METHOD PUBLIC PreExecutionCheck
VAR_INPUT
	Check : I_PreExecutionChecks;
END_VAR
Check.IsTrue(ipSrcImage.IsValid, 'ipSrcImage must contain an image');
Check.IsTrue(ipSrcImage.HasChannelCount(1), 'ipSrcImage must have 1 channel');
Check.IsTrue(ipSrcImage.IsPixelDepth(8), 'ipSrcImage must have 8 bit pixel depth');
Check.IsTrue((fMaxValue.Value >= 0.0), 'fMaxValue must be greater than or equal to 0');
Check.IsTrue((fMaxValue.Value <= 255.0), 'fMaxValue must be less than or equal to 255');
Check.IsTrue((eThresholdType.Value = ETcVnThresholdType.TCVN_TT_BINARY OR 
              eThresholdType.Value = ETcVnThresholdType.TCVN_TT_BINARY_INV), 'eThresholdType must be TCVN_TT_BINARY or TCVN_TT_BINARY_INV');
Check.IsTrue(nBlockSize.Value >= 3, 'nBlockSize must be greater than or equal to 3');
Check.IsTrue(nBlockSize.IsOdd, 'nBlockSize must be an odd number');
END_METHOD

END_FUNCTION_BLOCK

// ---- Nodes/Image Segmentation/Node_F_VN_SauvolaThreshold.TcPOU
{attribute 'linkalways'} 
{attribute 'no_explicit_call' := 'This FB is a CLASS and must be accessed using methods or properties'}
{attribute 'enable_dynamic_creation'}
FUNCTION_BLOCK Node_F_VN_SauvolaThreshold EXTENDS VisionNode
VAR
	ipSrcImage : _ITcVnImage;
    pipDestImage : _ITcVnImage;
    nBlockSize : _UDINT(3);
    fParamK : _LREAL(0.0);
    fMaxSigma : _LREAL(0.0);
    eThresholdType : _ETcVnThresholdType(ETcVnThresholdType.TCVN_TT_BINARY);
    hrPrev : _HRESULT(S_OK);
	hresult : _HRESULT(S_OK);
END_VAR

METHOD PUBLIC  Clone : I_Node
VAR
	pNode : POINTER TO Node_F_VN_SauvolaThreshold;
END_VAR
pNode := __NEW(Node_F_VN_SauvolaThreshold);
Clone := pNode^;
END_METHOD

METHOD FB_init : BOOL
VAR_INPUT
	bInitRetains : BOOL; // if TRUE, the retain variables are initialized (warm start / cold start)
	bInCopyCode : BOOL;  // if TRUE, the instance afterwards gets moved into the copy code (online change)
END_VAR
AddInput('ipSrcImage', ipSrcImage);
AddParameter('nBlockSize', nBlockSize);
AddParameter('fParamK', fParamK);
AddParameter('fMaxSigma', fMaxSigma);
AddParameter('eThresholdType', eThresholdType);
AddInput('hrPrev', hrPrev);
AddOutput('pipDestImage', pipDestImage);
AddOutput('hresult', hresult);
END_METHOD

METHOD PROTECTED OnExecute
hresult.Value := F_VN_SauvolaThreshold(
	ipSrcImage := ipSrcImage.Value,
	pipDestImage := pipDestImage.Value,
    nBlockSize := nBlockSize.Value,
    fParamK := fParamK.Value,
    fMaxSigma := fMaxSigma.Value,
    eThresholdType := eThresholdType.Value,
	hrPrev := hrPrev.Value);
END_METHOD

METHOD PUBLIC PreExecutionCheck
VAR_INPUT
	Check : I_PreExecutionChecks;
END_VAR
Check.IsTrue(ipSrcImage.IsValid, 'ipSrcImage must contain an image');
Check.IsTrue(ipSrcImage.HasChannelCount(1), 'ipSrcImage must have 1 channel');

Check.IsTrue((ipSrcImage.IsPixelDepth(8) OR
              ipSrcImage.IsPixelDepth(16) OR
              ipSrcImage.IsPixelDepth(32) OR
              ipSrcImage.IsPixelDepth(6432)), 'ipSrcImage must have 8, 16, 32, or 64 bit pixel depth');

Check.IsTrue(nBlockSize.IsOdd, 'nBlockSize must be an odd number');
Check.IsTrue(nBlockSize.Value >= 3, 'nBlockSize must be greater than or equal to 3');

Check.IsTrue((fParamK.Value >= 0.0), 'fMaxValue must be greater than or equal to 0');
Check.IsTrue((fParamK.Value <= 1.0), 'fMaxValue must be less than or equal to 1');

Check.IsTrue((fMaxSigma.Value >= 0.0), 'fMaxValue must be greater than or equal to 0');

Check.IsTrue((eThresholdType.Value = ETcVnThresholdType.TCVN_TT_BINARY OR 
              eThresholdType.Value = ETcVnThresholdType.TCVN_TT_BINARY_INV), 'eThresholdType must be TCVN_TT_BINARY or TCVN_TT_BINARY_INV');
END_METHOD

END_FUNCTION_BLOCK

// ---- Nodes/Image Segmentation/Node_F_VN_DoubleThreshold.TcPOU
{attribute 'linkalways'} 
{attribute 'no_explicit_call' := 'This FB is a CLASS and must be accessed using methods or properties'}
{attribute 'enable_dynamic_creation'}
FUNCTION_BLOCK Node_F_VN_DoubleThreshold EXTENDS VisionNode
VAR
	ipSrcImage : _ITcVnImage;
    ipDestImage : _ITcVnImage;
    fLowThreshold : _LREAL(0.0);
    fHighThreshold : _LREAL(0.0);
    fMaxValue : _LREAL(0.0);
    hrPrev : _HRESULT(S_OK);
	hresult : _HRESULT(S_OK);
END_VAR

METHOD PUBLIC  Clone : I_Node
VAR
	pNode : POINTER TO Node_F_VN_DoubleThreshold;
END_VAR
pNode := __NEW(Node_F_VN_DoubleThreshold);
Clone := pNode^;
END_METHOD

METHOD FB_init : BOOL
VAR_INPUT
	bInitRetains : BOOL; // if TRUE, the retain variables are initialized (warm start / cold start)
	bInCopyCode : BOOL;  // if TRUE, the instance afterwards gets moved into the copy code (online change)
END_VAR
AddInput('ipSrcImage', ipSrcImage);
AddParameter('fLowThreshold', fLowThreshold);
AddParameter('fHighThreshold', fHighThreshold);
AddParameter('fMaxValue', fMaxValue);
AddInput('hrPrev', hrPrev);
AddOutput('ipDestImage', ipDestImage);
AddOutput('hresult', hresult);
END_METHOD

METHOD PROTECTED OnExecute
hresult.Value := F_VN_DoubleThreshold(
	ipSrcImage := ipSrcImage.Value,
	ipDestImage := ipDestImage.Value,
    fLowThreshold := fLowThreshold.Value,
    fHighThreshold := fHighThreshold.Value,
    fMaxValue := fMaxValue.Value,
	hrPrev := hrPrev.Value);
END_METHOD

METHOD PUBLIC PreExecutionCheck
VAR_INPUT
	Check : I_PreExecutionChecks;
END_VAR
VAR
    pixelFormat : TcVnPixelFormat;
END_VAR
Check.IsTrue(ipSrcImage.IsValid, 'ipSrcImage must contain an image');
Check.IsTrue(ipSrcImage.HasChannelCount(1), 'ipSrcImage must have 1 channel');
Check.IsTrue((ipSrcImage.IsPixelDepth(8) OR
              ipSrcImage.IsPixelDepth(16) OR
              ipSrcImage.IsPixelDepth(32) OR
              ipSrcImage.IsPixelDepth(64)), 'ipSrcImage must have 8, 16, 32, or 64 bit pixel depth');

ipSrcImage.TryGetPixelFormat(pixelFormat);
Check.IsTrue(IsMaxValueCompatibleWithPixelDepth(fMaxValue.Value, pixelFormat.nElementSize), 'fMaxValue is not compatible with pixel depth');
END_METHOD

END_FUNCTION_BLOCK

// ---- Nodes/Image Segmentation/Node_F_VN_WatershedSegmentationExp.TcPOU
{attribute 'linkalways'} 
{attribute 'no_explicit_call' := 'This FB is a CLASS and must be accessed using methods or properties'}
{attribute 'enable_dynamic_creation'}
FUNCTION_BLOCK Node_F_VN_WatershedSegmentationExp EXTENDS VisionNode
VAR
	ipSrcImage : _ITcVnImage;
    ipDestImage : _ITcVnImage;
    ipMarkers : _ITcVnImage;
    hrPrev : _HRESULT(S_OK);
	hresult : _HRESULT(S_OK);
END_VAR

METHOD PUBLIC  Clone : I_Node
VAR
	pNode : POINTER TO Node_F_VN_WatershedSegmentationExp;
END_VAR
pNode := __NEW(Node_F_VN_WatershedSegmentationExp);
Clone := pNode^;
END_METHOD

METHOD FB_init : BOOL
VAR_INPUT
	bInitRetains : BOOL; // if TRUE, the retain variables are initialized (warm start / cold start)
	bInCopyCode : BOOL;  // if TRUE, the instance afterwards gets moved into the copy code (online change)
END_VAR
AddInput('ipSrcImage', ipSrcImage);
AddInput('ipMarkers', ipMarkers);
AddInput('hrPrev', hrPrev);
AddOutput('ipDestImage', ipDestImage);
AddOutput('hresult',hresult);
END_METHOD

METHOD PROTECTED OnExecute
hresult.Value := F_VN_WatershedSegmentationExp(
	ipSrcImage := ipSrcImage.Value,
	ipDestImage := ipDestImage.Value,
    ipMarkers := ipMarkers.Value,
	hrPrev := hrPrev.Value);
END_METHOD

METHOD PUBLIC PreExecutionCheck
VAR_INPUT
	Check : I_PreExecutionChecks;
END_VAR
Check.IsTrue(ipSrcImage.IsValid, 'ipSrcImage must contain an image');
Check.IsTrue(ipSrcImage.HasChannelCount(3), 'ipSrcImage must have 3 channels');
Check.IsTrue(ipSrcImage.IsPixelDepth(8), 'ipSrcImage must have 8 bit pixel depth');
Check.IsTrue(ipMarkers.IsValid, 'ipMarkers must contain an image');
Check.IsTrue(ipMarkers.HasChannelCount(1), 'ipMarkers must have 1 channel');
Check.IsTrue(ipMarkers.IsPixelDepth(32), 'ipMarkers must have DINT 32 bit pixel depth');
END_METHOD

END_FUNCTION_BLOCK

// ---- Nodes/Image Segmentation/Node_F_VN_CheckColorRange.TcPOU
{attribute 'linkalways'} 
{attribute 'no_explicit_call' := 'This FB is a CLASS and must be accessed using methods or properties'}
{attribute 'enable_dynamic_creation'}
FUNCTION_BLOCK Node_F_VN_CheckColorRange EXTENDS VisionNode
VAR
	ipSrcImage : _ITcVnImage;
    ipDestImage : _ITcVnImage;
    aLowerBounds : _TcVnVector4_LREAL;
    aUpperBounds : _TcVnVector4_LREAL;
    hrPrev : _HRESULT(S_OK);
	hresult : _HRESULT(S_OK);
END_VAR

METHOD PUBLIC  Clone : I_Node
VAR
	pNode : POINTER TO Node_F_VN_CheckColorRange;
END_VAR
pNode := __NEW(Node_F_VN_CheckColorRange);
Clone := pNode^;
END_METHOD

METHOD FB_init : BOOL
VAR_INPUT
	bInitRetains : BOOL; // if TRUE, the retain variables are initialized (warm start / cold start)
	bInCopyCode : BOOL;  // if TRUE, the instance afterwards gets moved into the copy code (online change)
END_VAR
AddInput('ipSrcImage', ipSrcImage);
AddInput('aLowerBounds', aLowerBounds);
AddInput('aUpperBounds', aUpperBounds);
AddInput('hrPrev', hrPrev);
AddOutput('ipDestImage', ipDestImage);
AddOutput('hresult', hresult);
END_METHOD

METHOD PROTECTED OnExecute
hresult.Value := F_VN_CheckColorRange(
	ipSrcImage := ipSrcImage.Value,
	ipDestImage := ipDestImage.Value,
    aLowerBounds := aLowerBounds.Value,
    aUpperBounds := aUpperBounds.Value,
	hrPrev := hrPrev.Value);
END_METHOD

METHOD PUBLIC PreExecutionCheck
VAR_INPUT
	Check : I_PreExecutionChecks;
END_VAR
Check.IsTrue(ipSrcImage.IsValid, 'ipSrcImage must contain an image');
END_METHOD

END_FUNCTION_BLOCK

// ---- Nodes/Image Segmentation/Node_F_VN_AdaptiveThreshold.TcPOU
{attribute 'linkalways'} 
{attribute 'no_explicit_call' := 'This FB is a CLASS and must be accessed using methods or properties'}
{attribute 'enable_dynamic_creation'}
FUNCTION_BLOCK Node_F_VN_AdaptiveThreshold EXTENDS VisionNode
VAR
	ipSrcImage : _ITcVnImage;
    ipDestImage : _ITcVnImage;
    fMaxValue : _LREAL(0.0);
    hrPrev : _HRESULT(S_OK);
	hresult : _HRESULT(S_OK);
END_VAR

METHOD PUBLIC  Clone : I_Node
VAR
	pNode : POINTER TO Node_F_VN_AdaptiveThreshold;
END_VAR
pNode := __NEW(Node_F_VN_AdaptiveThreshold);
Clone := pNode^;
END_METHOD

METHOD FB_init : BOOL
VAR_INPUT
	bInitRetains : BOOL; // if TRUE, the retain variables are initialized (warm start / cold start)
	bInCopyCode : BOOL;  // if TRUE, the instance afterwards gets moved into the copy code (online change)
END_VAR
AddInput('ipSrcImage', ipSrcImage);
AddParameter('fMaxValue', fMaxValue);
AddInput('hrPrev', hrPrev);
AddOutput('ipDestImage', ipDestImage);
AddOutput('hresult', hresult);
END_METHOD

METHOD PROTECTED OnExecute
hresult.Value := F_VN_AdaptiveThreshold(
	ipSrcImage := ipSrcImage.Value,
	ipDestImage := ipDestImage.Value,
    fMaxValue := fMaxValue.Value,
	hrPrev := hrPrev.Value);
END_METHOD

METHOD PUBLIC PreExecutionCheck
VAR_INPUT
	Check : I_PreExecutionChecks;
END_VAR
Check.IsTrue(ipSrcImage.IsValid, 'ipSrcImage must contain an image');
Check.IsTrue(ipSrcImage.HasChannelCount(1), 'ipSrcImage must have 1 channel');
Check.IsTrue(ipSrcImage.IsPixelDepth(8), 'ipSrcImage must have 8 bit pixel depth');
Check.IsTrue((fMaxValue.Value >= 0.0), 'fMaxValue must be greater than or equal to 0');
Check.IsTrue((fMaxValue.Value <= 255.0), 'fMaxValue must be less than or equal to 255');
END_METHOD

END_FUNCTION_BLOCK

// ---- Nodes/Image Segmentation/Node_F_VN_Threshold.TcPOU
{attribute 'linkalways'} 
{attribute 'no_explicit_call' := 'This FB is a CLASS and must be accessed using methods or properties'}
{attribute 'enable_dynamic_creation'}
FUNCTION_BLOCK Node_F_VN_Threshold EXTENDS VisionNode
VAR
	ipSrcImage : _ITcVnImage;
    ipDestImage : _ITcVnImage;
    fThreshold : _LREAL(0.0);
    fMaxValue : _LREAL(0.0);
	eThresholdType : _ETcVnThresholdType(ETcVnThresholdType.TCVN_TT_BINARY);
    hrPrev : _HRESULT(S_OK);
	hresult : _HRESULT(S_OK);
END_VAR

METHOD PUBLIC  Clone : I_Node
VAR
	pNode : POINTER TO Node_F_VN_Threshold;
END_VAR
pNode := __NEW(Node_F_VN_Threshold);
Clone := pNode^;
END_METHOD

METHOD FB_init : BOOL
VAR_INPUT
	bInitRetains : BOOL; // if TRUE, the retain variables are initialized (warm start / cold start)
	bInCopyCode : BOOL;  // if TRUE, the instance afterwards gets moved into the copy code (online change)
END_VAR
AddInput('ipSrcImage', ipSrcImage);
AddParameter('fThreshold', fThreshold);
AddParameter('fMaxValue', fMaxValue);
AddParameter('eThresholdType', eThresholdType);
AddInput('hrPrev', hrPrev);
AddOutput('ipDestImage', ipDestImage);
AddOutput('hresult',hresult);
END_METHOD

METHOD PROTECTED OnExecute
hresult.Value := F_VN_Threshold(
	ipSrcImage := ipSrcImage.Value, 
	ipDestImage := ipDestImage.Value, 
	fThreshold := fThreshold.Value, 
	fMaxValue := fMaxValue.Value, 
	eThresholdType := eThresholdType.Value, 
	hrPrev := hrPrev.Value);
END_METHOD

METHOD PUBLIC PreExecutionCheck
VAR_INPUT
	Check : I_PreExecutionChecks;
END_VAR
VAR
    dynamicThresholding : BOOL;
    pixelFormat : TcVnPixelFormat;
END_VAR
Check.IsTrue(ipSrcImage.IsValid, 'ipSrcImage must contain an image');

CASE eThresholdType.Value OF
    TCVN_TT_OTSU_BINARY,
    TCVN_TT_OTSU_BINARY_INV,
    TCVN_TT_OTSU_TRUNC,
    TCVN_TT_OTSU_TOZERO,
    TCVN_TT_OTSU_TOZERO_INV,
    TCVN_TT_TRIANGLE_BINARY,
    TCVN_TT_TRIANGLE_BINARY_INV,
    TCVN_TT_TRIANGLE_TRUNC,
    TCVN_TT_TRIANGLE_TOZERO,
    TCVN_TT_TRIANGLE_TOZERO_INV :
        dynamicThresholding := TRUE;
END_CASE

IF dynamicThresholding THEN
    Check.IsTrue(ipSrcImage.HasChannelCount(1), 'ipSrcImage must have 1 channel when using dynamic thresholding');
    Check.IsTrue(ipSrcImage.IsPixelDepth(8), 'ipSrcImage must have 8 bit pixel depth when using dynamic thresholding');
ELSE
    Check.IsTrue((ipSrcImage.HasChannelCount(1) OR ipSrcImage.HasChannelCount(3)), 'ipSrcImage must have 1 or 3 channels');
END_IF

ipSrcImage.TryGetPixelFormat(pixelFormat);
Check.IsTrue(IsMaxValueCompatibleWithPixelDepth(fMaxValue.Value, pixelFormat.nElementSize), 'fMaxValue is not compatible with pixel depth');
END_METHOD

END_FUNCTION_BLOCK

// ---- Nodes/Keypoint Features/Node_F_VN_FilterGoodMatches.TcPOU
{attribute 'linkalways'} 
{attribute 'no_explicit_call' := 'This FB is a CLASS and must be accessed using methods or properties'}
{attribute 'enable_dynamic_creation'}
FUNCTION_BLOCK Node_F_VN_FilterGoodMatches EXTENDS VisionNode
VAR
    ipMatches : _ITcVnContainer;
    ipGoodMatches : _ITcVnContainer;
    fMaxDist : _REAL(0.0);
    fMaxKnnRatio : _REAL(0.0);
    hrPrev : _HRESULT(S_OK);
	hresult : _HRESULT(S_OK);
END_VAR

METHOD PUBLIC  Clone : I_Node
VAR
	pNode : POINTER TO Node_F_VN_FilterGoodMatches;
END_VAR
pNode := __NEW(Node_F_VN_FilterGoodMatches);
Clone := pNode^;
END_METHOD

METHOD FB_init : BOOL
VAR_INPUT
	bInitRetains : BOOL; // if TRUE, the retain variables are initialized (warm start / cold start)
	bInCopyCode : BOOL;  // if TRUE, the instance afterwards gets moved into the copy code (online change)
END_VAR
AddInput('ipMatches', ipMatches);
AddParameter('fMaxDist', fMaxDist);
AddParameter('fMaxKnnRatio', fMaxKnnRatio);
AddInput('hrPrev', hrPrev);
AddOutput('ipGoodMatches', ipGoodMatches);
AddOutput('hresult',hresult);
END_METHOD

METHOD PROTECTED OnExecute
hresult.Value := F_VN_FilterGoodMatches(
    ipMatches := ipMatches.Value,
    ipGoodMatches := ipGoodMatches.Value,
    fMaxDist := fMaxDist.Value,
    fMaxKnnRatio := fMaxKnnRatio.Value,
	hrPrev:= hrPrev.Value);
END_METHOD

METHOD PUBLIC PreExecutionCheck
VAR_INPUT
	Check : I_PreExecutionChecks;
END_VAR
Check.IsTrue(ipMatches.IsValid, 'ipMatches must be a valid container');
Check.IsTrue((ipMatches.IsType(TC_GLOBAL_CONST_LIST.ContainerType_Vector_TcVnDMatch) OR
              ipMatches.IsType(TC_GLOBAL_CONST_LIST.ContainerType_Vector_Vector_TcVnDMatch)),
              'ipMatches contains incorrect type');
              
IF NOT (fMaxDist.Value = -1) THEN
    Check.IsTrue(fMaxDist.Value >= 0, 'fMaxDist must be greater than or equal to 0');
END_IF

IF NOT (fMaxKnnRatio.Value = -1) THEN
    Check.IsTrue((fMaxKnnRatio.Value >= 0 OR fMaxDist.Value <= 1), 'fMaxDist must be within 0 to 1');
END_IF
END_METHOD

END_FUNCTION_BLOCK

// ---- Nodes/Keypoint Features/Node_F_VN_FindReferenceKeyPointsInImage.TcPOU
{attribute 'linkalways'}
{attribute 'no_explicit_call' := 'This FB is a CLASS and must be accessed using methods or properties'}
{attribute 'enable_dynamic_creation'}
FUNCTION_BLOCK Node_F_VN_FindReferenceKeyPointsInImage EXTENDS VisionNode
VAR
    ipSrcKeyPoints : _ITcVnContainer;
    ipSrcDescriptors : _ITcVnImage;
    ipRefKeyPoints : _ITcVnContainer;
    ipRefDescriptors : _ITcVnImage;
    nRefImageWidth : _UDINT(0);
    nRefImageHeight : _UDINT(0);
    ipEdgePoints : _ITcVnContainer;
    fMaxDist : _REAL(-1.0);
    fMaxKnnRatio : _REAL(-1.0);
    eNormType : _ETcVnNormalizationType(ETcVnNormalizationType.TCVN_NT_HAMMING);
    hrPrev : _HRESULT(S_OK);
    aPerspectiveTransform : _TcVnMatrix3x3_LREAL;
    nNumberOfGoodMatches : _UDINT(0);
    nNumberOfInliers : _UDINT(0);
    hresult : _HRESULT(S_OK);
END_VAR

METHOD PUBLIC Clone : I_Node
VAR
    pNode : POINTER TO Node_F_VN_FindReferenceKeyPointsInImage;
END_VAR
pNode := __NEW(Node_F_VN_FindReferenceKeyPointsInImage);
Clone := pNode^;
END_METHOD

METHOD FB_init : BOOL
VAR_INPUT
    bInitRetains : BOOL;
    bInCopyCode : BOOL;
END_VAR
AddInput('ipSrcKeyPoints', ipSrcKeyPoints);
AddInput('ipSrcDescriptors', ipSrcDescriptors);
AddInput('ipRefKeyPoints', ipRefKeyPoints);
AddInput('ipRefDescriptors', ipRefDescriptors);
AddInput('nRefImageWidth', nRefImageWidth);
AddInput('nRefImageHeight', nRefImageHeight);
AddOutput('ipEdgePoints', ipEdgePoints);
AddParameter('fMaxDist', fMaxDist);
AddParameter('fMaxKnnRatio', fMaxKnnRatio);
AddParameter('eNormType', eNormType);
AddInput('hrPrev', hrPrev);
AddOutput('aPerspectiveTransform', aPerspectiveTransform);
AddOutput('nNumberOfGoodMatches', nNumberOfGoodMatches);
AddOutput('nNumberOfInliers', nNumberOfInliers);
AddOutput('hresult', hresult);
END_METHOD

METHOD PROTECTED OnExecute
VAR
    perspectiveTransform : TcVnMatrix3x3_LREAL;
    numberOfGoodMatches : UDINT;
    numberOfInliers : UDINT;
END_VAR
hresult.Value := F_VN_FindReferenceKeyPointsInImage(
    ipSrcKeyPoints := ipSrcKeyPoints.Value,
    ipSrcDescriptors := ipSrcDescriptors.Value,
    ipRefKeyPoints := ipRefKeyPoints.Value,
    ipRefDescriptors := ipRefDescriptors.Value,
    nRefImageWidth := nRefImageWidth.Value,
    nRefImageHeight := nRefImageHeight.Value,
    ipEdgePoints := ipEdgePoints.Value,
    fMaxDist := fMaxDist.Value,
    fMaxKnnRatio := fMaxKnnRatio.Value,
    eNormType := eNormType.Value,
    hrPrev := hrPrev.Value,
    aPerspectiveTransform => perspectiveTransform,
    nNumberOfGoodMatches => numberOfGoodMatches,
    nNumberOfInliers => numberOfInliers);

aPerspectiveTransform.Value := perspectiveTransform;
nNumberOfGoodMatches.Value := numberOfGoodMatches;
nNumberOfInliers.Value := numberOfInliers;
END_METHOD

METHOD PUBLIC PreExecutionCheck
VAR_INPUT
    Check : I_PreExecutionChecks;
END_VAR
Check.IsTrue(ipSrcKeyPoints.IsValid, 'ipSrcKeyPoints must contain a container');
Check.IsTrue(ipSrcDescriptors.IsValid, 'ipSrcDescriptors must contain an image');
Check.IsTrue(ImagesHaveMatchingPixelFormats(ipSrcDescriptors.Value, ipRefDescriptors.Value), 'Source and reference descriptors must have matching pixel formats');
Check.IsTrue(IsImage1WidthEqualToImage2Width(ipSrcDescriptors.Value, ipRefDescriptors.Value), 'Source and reference descriptors must have matching descriptor lengths');
Check.IsTrue(ipRefKeyPoints.IsValid, 'ipRefKeyPoints must contain a container');
Check.IsTrue(ipRefDescriptors.IsValid, 'ipRefDescriptors must contain an image');
Check.IsTrue(nRefImageWidth.Value > 0, 'nRefImageWidth must be greater than 0');
Check.IsTrue(nRefImageHeight.Value > 0, 'nRefImageHeight must be greater than 0');
Check.IsTrue((fMaxDist.Value = -1.0) OR (fMaxDist.Value >= 0.0), 'fMaxDist must be -1 to disable the filter, or at least 0');
Check.IsTrue((fMaxKnnRatio.Value = -1.0) OR
             ((fMaxKnnRatio.Value >= 0.0) AND (fMaxKnnRatio.Value <= 1.0)), 'fMaxKnnRatio must be -1 to disable the filter, or between 0 and 1');
Check.IsTrue((eNormType.Value = ETcVnNormalizationType.TCVN_NT_L1) OR
             (eNormType.Value = ETcVnNormalizationType.TCVN_NT_L2) OR
             (eNormType.Value = ETcVnNormalizationType.TCVN_NT_L2SQR) OR
             (eNormType.Value = ETcVnNormalizationType.TCVN_NT_HAMMING) OR
             (eNormType.Value = ETcVnNormalizationType.TCVN_NT_HAMMING2), 'Unsupported eNormType');
END_METHOD

END_FUNCTION_BLOCK

// ---- Nodes/Keypoint Features/Node_F_VN_FindReferenceKeyPointsInImageExp.TcPOU
{attribute 'linkalways'}
{attribute 'no_explicit_call' := 'This FB is a CLASS and must be accessed using methods or properties'}
{attribute 'enable_dynamic_creation'}
FUNCTION_BLOCK Node_F_VN_FindReferenceKeyPointsInImageExp EXTENDS VisionNode
VAR
    ipSrcKeyPoints : _ITcVnContainer;
    ipSrcDescriptors : _ITcVnImage;
    ipRefKeyPoints : _ITcVnContainer;
    ipRefDescriptors : _ITcVnImage;
    nRefImageWidth : _UDINT(0);
    nRefImageHeight : _UDINT(0);
    ipEdgePoints : _ITcVnContainer;
    fMaxDist : _REAL(-1.0);
    fMaxKnnRatio : _REAL(-1.0);
    eNormType : _ETcVnNormalizationType(ETcVnNormalizationType.TCVN_NT_HAMMING);
    eAlgorithm : _ETcVnEstimationAlgorithm(ETcVnEstimationAlgorithm.TCVN_EA_RANSAC);
    fReprojThreshold : _LREAL(3.0);
    nMaxIterations : _UDINT(2000);
    fConfidence : _LREAL(0.995);
    ipGoodMatches : _ITcVnContainer;
    ipInlierMask : _ITcVnContainer;
    hrPrev : _HRESULT(S_OK);
    aPerspectiveTransform : _TcVnMatrix3x3_LREAL;
    nNumberOfGoodMatches : _UDINT(0);
    nNumberOfInliers : _UDINT(0);
    hresult : _HRESULT(S_OK);
END_VAR

METHOD PUBLIC Clone : I_Node
VAR
    pNode : POINTER TO Node_F_VN_FindReferenceKeyPointsInImageExp;
END_VAR
pNode := __NEW(Node_F_VN_FindReferenceKeyPointsInImageExp);
Clone := pNode^;
END_METHOD

METHOD FB_init : BOOL
VAR_INPUT
    bInitRetains : BOOL;
    bInCopyCode : BOOL;
END_VAR
AddInput('ipSrcKeyPoints', ipSrcKeyPoints);
AddInput('ipSrcDescriptors', ipSrcDescriptors);
AddInput('ipRefKeyPoints', ipRefKeyPoints);
AddInput('ipRefDescriptors', ipRefDescriptors);
AddInput('nRefImageWidth', nRefImageWidth);
AddInput('nRefImageHeight', nRefImageHeight);
AddOutput('ipEdgePoints', ipEdgePoints);
AddParameter('fMaxDist', fMaxDist);
AddParameter('fMaxKnnRatio', fMaxKnnRatio);
AddParameter('eNormType', eNormType);
AddParameter('eAlgorithm', eAlgorithm);
AddParameter('fReprojThreshold', fReprojThreshold);
AddParameter('nMaxIterations', nMaxIterations);
AddParameter('fConfidence', fConfidence);
AddOutput('ipGoodMatches', ipGoodMatches);
AddOutput('ipInlierMask', ipInlierMask);
AddInput('hrPrev', hrPrev);
AddOutput('aPerspectiveTransform', aPerspectiveTransform);
AddOutput('nNumberOfGoodMatches', nNumberOfGoodMatches);
AddOutput('nNumberOfInliers', nNumberOfInliers);
AddOutput('hresult', hresult);
END_METHOD

METHOD PROTECTED OnExecute
VAR
    perspectiveTransform : TcVnMatrix3x3_LREAL;
    numberOfGoodMatches : UDINT;
    numberOfInliers : UDINT;
END_VAR
hresult.Value := F_VN_FindReferenceKeyPointsInImageExp(
    ipSrcKeyPoints := ipSrcKeyPoints.Value,
    ipSrcDescriptors := ipSrcDescriptors.Value,
    ipRefKeyPoints := ipRefKeyPoints.Value,
    ipRefDescriptors := ipRefDescriptors.Value,
    nRefImageWidth := nRefImageWidth.Value,
    nRefImageHeight := nRefImageHeight.Value,
    ipEdgePoints := ipEdgePoints.Value,
    fMaxDist := fMaxDist.Value,
    fMaxKnnRatio := fMaxKnnRatio.Value,
    eNormType := eNormType.Value,
    eAlgorithm := eAlgorithm.Value,
    fReprojThreshold := fReprojThreshold.Value,
    nMaxIterations := nMaxIterations.Value,
    fConfidence := fConfidence.Value,
    ipGoodMatches := ipGoodMatches.Value,
    ipInlierMask := ipInlierMask.Value,
    hrPrev := hrPrev.Value,
    aPerspectiveTransform => perspectiveTransform,
    nNumberOfGoodMatches => numberOfGoodMatches,
    nNumberOfInliers => numberOfInliers);

aPerspectiveTransform.Value := perspectiveTransform;
nNumberOfGoodMatches.Value := numberOfGoodMatches;
nNumberOfInliers.Value := numberOfInliers;
END_METHOD

METHOD PUBLIC PreExecutionCheck
VAR_INPUT
    Check : I_PreExecutionChecks;
END_VAR
Check.IsTrue(ipSrcKeyPoints.IsValid, 'ipSrcKeyPoints must contain a container');
Check.IsTrue(ipSrcDescriptors.IsValid, 'ipSrcDescriptors must contain an image');
Check.IsTrue(ImagesHaveMatchingPixelFormats(ipSrcDescriptors.Value, ipRefDescriptors.Value), 'Source and reference descriptors must have matching pixel formats');
Check.IsTrue(IsImage1WidthEqualToImage2Width(ipSrcDescriptors.Value, ipRefDescriptors.Value), 'Source and reference descriptors must have matching descriptor lengths');
Check.IsTrue(ipRefKeyPoints.IsValid, 'ipRefKeyPoints must contain a container');
Check.IsTrue(ipRefDescriptors.IsValid, 'ipRefDescriptors must contain an image');
Check.IsTrue(nRefImageWidth.Value > 0, 'nRefImageWidth must be greater than 0');
Check.IsTrue(nRefImageHeight.Value > 0, 'nRefImageHeight must be greater than 0');
Check.IsTrue((fMaxDist.Value = -1.0) OR (fMaxDist.Value >= 0.0), 'fMaxDist must be -1 to disable the filter, or at least 0');
Check.IsTrue((fMaxKnnRatio.Value = -1.0) OR
             ((fMaxKnnRatio.Value >= 0.0) AND (fMaxKnnRatio.Value <= 1.0)), 'fMaxKnnRatio must be -1 to disable the filter, or between 0 and 1');
Check.IsTrue((eNormType.Value = ETcVnNormalizationType.TCVN_NT_L1) OR
             (eNormType.Value = ETcVnNormalizationType.TCVN_NT_L2) OR
             (eNormType.Value = ETcVnNormalizationType.TCVN_NT_L2SQR) OR
             (eNormType.Value = ETcVnNormalizationType.TCVN_NT_HAMMING) OR
             (eNormType.Value = ETcVnNormalizationType.TCVN_NT_HAMMING2), 'Unsupported eNormType');
Check.IsTrue((eAlgorithm.Value = ETcVnEstimationAlgorithm.TCVN_EA_DEFAULT) OR
             (eAlgorithm.Value = ETcVnEstimationAlgorithm.TCVN_EA_LMEDS) OR
             (eAlgorithm.Value = ETcVnEstimationAlgorithm.TCVN_EA_RANSAC) OR
             (eAlgorithm.Value = ETcVnEstimationAlgorithm.TCVN_EA_RHO), 'Unsupported eAlgorithm');
// fReprojThreshold is only used by RANSAC and RHO.
Check.IsTrue(((eAlgorithm.Value <> ETcVnEstimationAlgorithm.TCVN_EA_RANSAC) AND
              (eAlgorithm.Value <> ETcVnEstimationAlgorithm.TCVN_EA_RHO)) OR
             (fReprojThreshold.Value > 0.0), 'fReprojThreshold must be greater than 0 for RANSAC and RHO');
Check.IsTrue(nMaxIterations.Value > 0, 'nMaxIterations must be greater than 0');
Check.IsTrue((fConfidence.Value > 0.0) AND (fConfidence.Value < 1.0), 'fConfidence must be between 0 and 1');
END_METHOD

END_FUNCTION_BLOCK

// ---- Nodes/Keypoint Features/Node_F_VN_FindReferenceKeyPointsInImageAKAZE.TcPOU
{attribute 'linkalways'}
{attribute 'no_explicit_call' := 'This FB is a CLASS and must be accessed using methods or properties'}
{attribute 'enable_dynamic_creation'}
FUNCTION_BLOCK Node_F_VN_FindReferenceKeyPointsInImageAKAZE EXTENDS VisionNode
VAR
    ipSrcImage : _ITcVnImage;
    ipRefKeyPoints : _ITcVnContainer;
    ipRefDescriptors : _ITcVnImage;
    nRefImageWidth : _UDINT(0);
    nRefImageHeight : _UDINT(0);
    ipEdgePoints : _ITcVnContainer;
    fMaxDist : _REAL(-1.0);
    fMaxKnnRatio : _REAL(-1.0);
    hrPrev : _HRESULT(S_OK);
    aPerspectiveTransform : _TcVnMatrix3x3_LREAL;
    nNumberOfGoodMatches : _UDINT(0);
    nNumberOfInliers : _UDINT(0);
    hresult : _HRESULT(S_OK);
END_VAR

METHOD PUBLIC Clone : I_Node
VAR
    pNode : POINTER TO Node_F_VN_FindReferenceKeyPointsInImageAKAZE;
END_VAR
pNode := __NEW(Node_F_VN_FindReferenceKeyPointsInImageAKAZE);
Clone := pNode^;
END_METHOD

METHOD FB_init : BOOL
VAR_INPUT
    bInitRetains : BOOL;
    bInCopyCode : BOOL;
END_VAR
AddInput('ipSrcImage', ipSrcImage);
AddInput('ipRefKeyPoints', ipRefKeyPoints);
AddInput('ipRefDescriptors', ipRefDescriptors);
AddInput('nRefImageWidth', nRefImageWidth);
AddInput('nRefImageHeight', nRefImageHeight);
AddOutput('ipEdgePoints', ipEdgePoints);
AddParameter('fMaxDist', fMaxDist);
AddParameter('fMaxKnnRatio', fMaxKnnRatio);
AddInput('hrPrev', hrPrev);
AddOutput('aPerspectiveTransform', aPerspectiveTransform);
AddOutput('nNumberOfGoodMatches', nNumberOfGoodMatches);
AddOutput('nNumberOfInliers', nNumberOfInliers);
AddOutput('hresult', hresult);
END_METHOD

METHOD PROTECTED OnExecute
VAR
    perspectiveTransform : TcVnMatrix3x3_LREAL;
    numberOfGoodMatches : UDINT;
    numberOfInliers : UDINT;
END_VAR
hresult.Value := F_VN_FindReferenceKeyPointsInImageAKAZE(
    ipSrcImage := ipSrcImage.Value,
    ipRefKeyPoints := ipRefKeyPoints.Value,
    ipRefDescriptors := ipRefDescriptors.Value,
    nRefImageWidth := nRefImageWidth.Value,
    nRefImageHeight := nRefImageHeight.Value,
    ipEdgePoints := ipEdgePoints.Value,
    fMaxDist := fMaxDist.Value,
    fMaxKnnRatio := fMaxKnnRatio.Value,
    hrPrev := hrPrev.Value,
    aPerspectiveTransform => perspectiveTransform,
    nNumberOfGoodMatches => numberOfGoodMatches,
    nNumberOfInliers => numberOfInliers);

aPerspectiveTransform.Value := perspectiveTransform;
nNumberOfGoodMatches.Value := numberOfGoodMatches;
nNumberOfInliers.Value := numberOfInliers;
END_METHOD

METHOD PUBLIC PreExecutionCheck
VAR_INPUT
    Check : I_PreExecutionChecks;
END_VAR
Check.IsTrue(ipSrcImage.IsValid, 'ipSrcImage must contain an image');
Check.IsTrue(ipSrcImage.HasChannelCount(1), 'ipSrcImage must have 1 channel');
Check.IsTrue(ipRefKeyPoints.IsValid, 'ipRefKeyPoints must contain a container');
Check.IsTrue(ipRefDescriptors.IsValid, 'ipRefDescriptors must contain an image');
Check.IsTrue(nRefImageWidth.Value > 0, 'nRefImageWidth must be greater than 0');
Check.IsTrue(nRefImageHeight.Value > 0, 'nRefImageHeight must be greater than 0');
Check.IsTrue((fMaxDist.Value = -1.0) OR (fMaxDist.Value >= 0.0), 'fMaxDist must be -1 to disable the filter, or at least 0');
Check.IsTrue((fMaxKnnRatio.Value = -1.0) OR
             ((fMaxKnnRatio.Value >= 0.0) AND (fMaxKnnRatio.Value <= 1.0)), 'fMaxKnnRatio must be -1 to disable the filter, or between 0 and 1');
END_METHOD

END_FUNCTION_BLOCK

// ---- Nodes/Keypoint Features/Node_F_VN_FindReferenceKeyPointsInImageAKAZEExp.TcPOU
{attribute 'linkalways'}
{attribute 'no_explicit_call' := 'This FB is a CLASS and must be accessed using methods or properties'}
{attribute 'enable_dynamic_creation'}
FUNCTION_BLOCK Node_F_VN_FindReferenceKeyPointsInImageAKAZEExp EXTENDS VisionNode
VAR
    ipSrcImage : _ITcVnImage;
    ipRefKeyPoints : _ITcVnContainer;
    ipRefDescriptors : _ITcVnImage;
    nRefImageWidth : _UDINT(0);
    nRefImageHeight : _UDINT(0);
    ipEdgePoints : _ITcVnContainer;
    fMaxDist : _REAL(-1.0);
    fMaxKnnRatio : _REAL(-1.0);
    eNormType : _ETcVnNormalizationType(ETcVnNormalizationType.TCVN_NT_HAMMING);
    ipSrcImageMask : _ITcVnImage;
    stAkazeParams : _TcVnParamsAKAZE;
    eAlgorithm : _ETcVnEstimationAlgorithm(ETcVnEstimationAlgorithm.TCVN_EA_RANSAC);
    fReprojThreshold : _LREAL(3.0);
    nMaxIterations : _UDINT(2000);
    fConfidence : _LREAL(0.995);
    hrPrev : _HRESULT(S_OK);
    aPerspectiveTransform : _TcVnMatrix3x3_LREAL;
    nNumberOfGoodMatches : _UDINT(0);
    nNumberOfInliers : _UDINT(0);
    hresult : _HRESULT(S_OK);
END_VAR

METHOD PUBLIC Clone : I_Node
VAR
    pNode : POINTER TO Node_F_VN_FindReferenceKeyPointsInImageAKAZEExp;
END_VAR
pNode := __NEW(Node_F_VN_FindReferenceKeyPointsInImageAKAZEExp);
Clone := pNode^;
END_METHOD

METHOD FB_init : BOOL
VAR_INPUT
    bInitRetains : BOOL;
    bInCopyCode : BOOL;
END_VAR
AddInput('ipSrcImage', ipSrcImage);
AddInput('ipRefKeyPoints', ipRefKeyPoints);
AddInput('ipRefDescriptors', ipRefDescriptors);
AddInput('nRefImageWidth', nRefImageWidth);
AddInput('nRefImageHeight', nRefImageHeight);
AddOutput('ipEdgePoints', ipEdgePoints);
AddParameter('fMaxDist', fMaxDist);
AddParameter('fMaxKnnRatio', fMaxKnnRatio);
AddParameter('eNormType', eNormType);
AddInput('ipSrcImageMask', ipSrcImageMask);
AddInput('stAkazeParams', stAkazeParams);
AddParameter('eAlgorithm', eAlgorithm);
AddParameter('fReprojThreshold', fReprojThreshold);
AddParameter('nMaxIterations', nMaxIterations);
AddParameter('fConfidence', fConfidence);
AddInput('hrPrev', hrPrev);
AddOutput('aPerspectiveTransform', aPerspectiveTransform);
AddOutput('nNumberOfGoodMatches', nNumberOfGoodMatches);
AddOutput('nNumberOfInliers', nNumberOfInliers);
AddOutput('hresult', hresult);
END_METHOD

METHOD PROTECTED OnExecute
VAR
    perspectiveTransform : TcVnMatrix3x3_LREAL;
    numberOfGoodMatches : UDINT;
    numberOfInliers : UDINT;
END_VAR
hresult.Value := F_VN_FindReferenceKeyPointsInImageAKAZEExp(
    ipSrcImage := ipSrcImage.Value,
    ipRefKeyPoints := ipRefKeyPoints.Value,
    ipRefDescriptors := ipRefDescriptors.Value,
    nRefImageWidth := nRefImageWidth.Value,
    nRefImageHeight := nRefImageHeight.Value,
    ipEdgePoints := ipEdgePoints.Value,
    fMaxDist := fMaxDist.Value,
    fMaxKnnRatio := fMaxKnnRatio.Value,
    eNormType := eNormType.Value,
    ipSrcImageMask := ipSrcImageMask.Value,
    stAkazeParams := stAkazeParams.Value,
    eAlgorithm := eAlgorithm.Value,
    fReprojThreshold := fReprojThreshold.Value,
    nMaxIterations := nMaxIterations.Value,
    fConfidence := fConfidence.Value,
    hrPrev := hrPrev.Value,
    aPerspectiveTransform => perspectiveTransform,
    nNumberOfGoodMatches => numberOfGoodMatches,
    nNumberOfInliers => numberOfInliers);

aPerspectiveTransform.Value := perspectiveTransform;
nNumberOfGoodMatches.Value := numberOfGoodMatches;
nNumberOfInliers.Value := numberOfInliers;
END_METHOD

METHOD PUBLIC PreExecutionCheck
VAR_INPUT
    Check : I_PreExecutionChecks;
END_VAR
Check.IsTrue(ipSrcImage.IsValid, 'ipSrcImage must contain an image');
Check.IsTrue(ipSrcImage.HasChannelCount(1), 'ipSrcImage must have 1 channel');
IF ipSrcImageMask.Value <> 0 THEN
    Check.IsTrue(ipSrcImageMask.IsValid, 'ipSrcImageMask must contain an image when connected');
    Check.IsTrue(IsImage1SizeEqualToImage2Size(ipSrcImage.Value, ipSrcImageMask.Value), 'ipSrcImageMask must have the same size as ipSrcImage');
END_IF
Check.IsTrue(ipRefKeyPoints.IsValid, 'ipRefKeyPoints must contain a container');
Check.IsTrue(ipRefDescriptors.IsValid, 'ipRefDescriptors must contain an image');
Check.IsTrue(nRefImageWidth.Value > 0, 'nRefImageWidth must be greater than 0');
Check.IsTrue(nRefImageHeight.Value > 0, 'nRefImageHeight must be greater than 0');
Check.IsTrue((fMaxDist.Value = -1.0) OR (fMaxDist.Value >= 0.0), 'fMaxDist must be -1 to disable the filter, or at least 0');
Check.IsTrue((fMaxKnnRatio.Value = -1.0) OR
             ((fMaxKnnRatio.Value >= 0.0) AND (fMaxKnnRatio.Value <= 1.0)), 'fMaxKnnRatio must be -1 to disable the filter, or between 0 and 1');
Check.IsTrue((eNormType.Value = ETcVnNormalizationType.TCVN_NT_L1) OR
             (eNormType.Value = ETcVnNormalizationType.TCVN_NT_L2) OR
             (eNormType.Value = ETcVnNormalizationType.TCVN_NT_L2SQR) OR
             (eNormType.Value = ETcVnNormalizationType.TCVN_NT_HAMMING) OR
             (eNormType.Value = ETcVnNormalizationType.TCVN_NT_HAMMING2), 'Unsupported eNormType');
IF ((stAkazeParams.Value.eDescrType = ETcVnFeatureDescriptorTypeAKAZE.TCVN_FDT_AKAZE_MLDB) OR
    (stAkazeParams.Value.eDescrType = ETcVnFeatureDescriptorTypeAKAZE.TCVN_FDT_AKAZE_MLDB_UPRIGHT)) THEN
    Check.IsTrue(stAkazeParams.Value.nDescrChannels = 3, 'nDescrChannels must be 3 when using AKAZE_MLDB');
END_IF
Check.IsTrue((eAlgorithm.Value = ETcVnEstimationAlgorithm.TCVN_EA_DEFAULT) OR
             (eAlgorithm.Value = ETcVnEstimationAlgorithm.TCVN_EA_LMEDS) OR
             (eAlgorithm.Value = ETcVnEstimationAlgorithm.TCVN_EA_RANSAC) OR
             (eAlgorithm.Value = ETcVnEstimationAlgorithm.TCVN_EA_RHO), 'Unsupported eAlgorithm');
// fReprojThreshold is only used by RANSAC and RHO.
Check.IsTrue(((eAlgorithm.Value <> ETcVnEstimationAlgorithm.TCVN_EA_RANSAC) AND
              (eAlgorithm.Value <> ETcVnEstimationAlgorithm.TCVN_EA_RHO)) OR
             (fReprojThreshold.Value > 0.0), 'fReprojThreshold must be greater than 0 for RANSAC and RHO');
Check.IsTrue(nMaxIterations.Value > 0, 'nMaxIterations must be greater than 0');
Check.IsTrue((fConfidence.Value > 0.0) AND (fConfidence.Value < 1.0), 'fConfidence must be between 0 and 1');
END_METHOD

END_FUNCTION_BLOCK

// ---- Nodes/Keypoint Features/Node_F_VN_FindReferenceKeyPointsInImageBRISK.TcPOU
{attribute 'linkalways'}
{attribute 'no_explicit_call' := 'This FB is a CLASS and must be accessed using methods or properties'}
{attribute 'enable_dynamic_creation'}
FUNCTION_BLOCK Node_F_VN_FindReferenceKeyPointsInImageBRISK EXTENDS VisionNode
VAR
    ipSrcImage : _ITcVnImage;
    ipRefKeyPoints : _ITcVnContainer;
    ipRefDescriptors : _ITcVnImage;
    nRefImageWidth : _UDINT(0);
    nRefImageHeight : _UDINT(0);
    ipEdgePoints : _ITcVnContainer;
    fMaxDist : _REAL(-1.0);
    fMaxKnnRatio : _REAL(-1.0);
    hrPrev : _HRESULT(S_OK);
    aPerspectiveTransform : _TcVnMatrix3x3_LREAL;
    nNumberOfGoodMatches : _UDINT(0);
    nNumberOfInliers : _UDINT(0);
    hresult : _HRESULT(S_OK);
END_VAR

METHOD PUBLIC Clone : I_Node
VAR
    pNode : POINTER TO Node_F_VN_FindReferenceKeyPointsInImageBRISK;
END_VAR
pNode := __NEW(Node_F_VN_FindReferenceKeyPointsInImageBRISK);
Clone := pNode^;
END_METHOD

METHOD FB_init : BOOL
VAR_INPUT
    bInitRetains : BOOL;
    bInCopyCode : BOOL;
END_VAR
AddInput('ipSrcImage', ipSrcImage);
AddInput('ipRefKeyPoints', ipRefKeyPoints);
AddInput('ipRefDescriptors', ipRefDescriptors);
AddInput('nRefImageWidth', nRefImageWidth);
AddInput('nRefImageHeight', nRefImageHeight);
AddOutput('ipEdgePoints', ipEdgePoints);
AddParameter('fMaxDist', fMaxDist);
AddParameter('fMaxKnnRatio', fMaxKnnRatio);
AddInput('hrPrev', hrPrev);
AddOutput('aPerspectiveTransform', aPerspectiveTransform);
AddOutput('nNumberOfGoodMatches', nNumberOfGoodMatches);
AddOutput('nNumberOfInliers', nNumberOfInliers);
AddOutput('hresult', hresult);
END_METHOD

METHOD PROTECTED OnExecute
VAR
    perspectiveTransform : TcVnMatrix3x3_LREAL;
    numberOfGoodMatches : UDINT;
    numberOfInliers : UDINT;
END_VAR
hresult.Value := F_VN_FindReferenceKeyPointsInImageBRISK(
    ipSrcImage := ipSrcImage.Value,
    ipRefKeyPoints := ipRefKeyPoints.Value,
    ipRefDescriptors := ipRefDescriptors.Value,
    nRefImageWidth := nRefImageWidth.Value,
    nRefImageHeight := nRefImageHeight.Value,
    ipEdgePoints := ipEdgePoints.Value,
    fMaxDist := fMaxDist.Value,
    fMaxKnnRatio := fMaxKnnRatio.Value,
    hrPrev := hrPrev.Value,
    aPerspectiveTransform => perspectiveTransform,
    nNumberOfGoodMatches => numberOfGoodMatches,
    nNumberOfInliers => numberOfInliers);

aPerspectiveTransform.Value := perspectiveTransform;
nNumberOfGoodMatches.Value := numberOfGoodMatches;
nNumberOfInliers.Value := numberOfInliers;
END_METHOD

METHOD PUBLIC PreExecutionCheck
VAR_INPUT
    Check : I_PreExecutionChecks;
END_VAR
Check.IsTrue(ipSrcImage.IsValid, 'ipSrcImage must contain an image');
Check.IsTrue(ipSrcImage.HasChannelCount(1), 'ipSrcImage must have 1 channel');
Check.IsTrue(ipRefKeyPoints.IsValid, 'ipRefKeyPoints must contain a container');
Check.IsTrue(ipRefDescriptors.IsValid, 'ipRefDescriptors must contain an image');
Check.IsTrue(nRefImageWidth.Value > 0, 'nRefImageWidth must be greater than 0');
Check.IsTrue(nRefImageHeight.Value > 0, 'nRefImageHeight must be greater than 0');
Check.IsTrue((fMaxDist.Value = -1.0) OR (fMaxDist.Value >= 0.0), 'fMaxDist must be -1 to disable the filter, or at least 0');
Check.IsTrue((fMaxKnnRatio.Value = -1.0) OR
             ((fMaxKnnRatio.Value >= 0.0) AND (fMaxKnnRatio.Value <= 1.0)), 'fMaxKnnRatio must be -1 to disable the filter, or between 0 and 1');
END_METHOD

END_FUNCTION_BLOCK

// ---- Nodes/Keypoint Features/Node_F_VN_FindReferenceKeyPointsInImageBRISKExp.TcPOU
{attribute 'linkalways'}
{attribute 'no_explicit_call' := 'This FB is a CLASS and must be accessed using methods or properties'}
{attribute 'enable_dynamic_creation'}
FUNCTION_BLOCK Node_F_VN_FindReferenceKeyPointsInImageBRISKExp EXTENDS VisionNode
VAR
    ipSrcImage : _ITcVnImage;
    ipRefKeyPoints : _ITcVnContainer;
    ipRefDescriptors : _ITcVnImage;
    nRefImageWidth : _UDINT(0);
    nRefImageHeight : _UDINT(0);
    ipEdgePoints : _ITcVnContainer;
    fMaxDist : _REAL(-1.0);
    fMaxKnnRatio : _REAL(-1.0);
    eNormType : _ETcVnNormalizationType(ETcVnNormalizationType.TCVN_NT_HAMMING);
    ipSrcImageMask : _ITcVnImage;
    stBriskParams : _TcVnParamsBRISK;
    eAlgorithm : _ETcVnEstimationAlgorithm(ETcVnEstimationAlgorithm.TCVN_EA_RANSAC);
    fReprojThreshold : _LREAL(3.0);
    nMaxIterations : _UDINT(2000);
    fConfidence : _LREAL(0.995);
    hrPrev : _HRESULT(S_OK);
    aPerspectiveTransform : _TcVnMatrix3x3_LREAL;
    nNumberOfGoodMatches : _UDINT(0);
    nNumberOfInliers : _UDINT(0);
    hresult : _HRESULT(S_OK);
END_VAR

METHOD PUBLIC Clone : I_Node
VAR
    pNode : POINTER TO Node_F_VN_FindReferenceKeyPointsInImageBRISKExp;
END_VAR
pNode := __NEW(Node_F_VN_FindReferenceKeyPointsInImageBRISKExp);
Clone := pNode^;
END_METHOD

METHOD FB_init : BOOL
VAR_INPUT
    bInitRetains : BOOL;
    bInCopyCode : BOOL;
END_VAR
AddInput('ipSrcImage', ipSrcImage);
AddInput('ipRefKeyPoints', ipRefKeyPoints);
AddInput('ipRefDescriptors', ipRefDescriptors);
AddInput('nRefImageWidth', nRefImageWidth);
AddInput('nRefImageHeight', nRefImageHeight);
AddOutput('ipEdgePoints', ipEdgePoints);
AddParameter('fMaxDist', fMaxDist);
AddParameter('fMaxKnnRatio', fMaxKnnRatio);
AddParameter('eNormType', eNormType);
AddInput('ipSrcImageMask', ipSrcImageMask);
AddInput('stBriskParams', stBriskParams);
AddParameter('eAlgorithm', eAlgorithm);
AddParameter('fReprojThreshold', fReprojThreshold);
AddParameter('nMaxIterations', nMaxIterations);
AddParameter('fConfidence', fConfidence);
AddInput('hrPrev', hrPrev);
AddOutput('aPerspectiveTransform', aPerspectiveTransform);
AddOutput('nNumberOfGoodMatches', nNumberOfGoodMatches);
AddOutput('nNumberOfInliers', nNumberOfInliers);
AddOutput('hresult', hresult);
END_METHOD

METHOD PROTECTED OnExecute
VAR
    perspectiveTransform : TcVnMatrix3x3_LREAL;
    numberOfGoodMatches : UDINT;
    numberOfInliers : UDINT;
END_VAR
hresult.Value := F_VN_FindReferenceKeyPointsInImageBRISKExp(
    ipSrcImage := ipSrcImage.Value,
    ipRefKeyPoints := ipRefKeyPoints.Value,
    ipRefDescriptors := ipRefDescriptors.Value,
    nRefImageWidth := nRefImageWidth.Value,
    nRefImageHeight := nRefImageHeight.Value,
    ipEdgePoints := ipEdgePoints.Value,
    fMaxDist := fMaxDist.Value,
    fMaxKnnRatio := fMaxKnnRatio.Value,
    eNormType := eNormType.Value,
    ipSrcImageMask := ipSrcImageMask.Value,
    stBriskParams := stBriskParams.Value,
    eAlgorithm := eAlgorithm.Value,
    fReprojThreshold := fReprojThreshold.Value,
    nMaxIterations := nMaxIterations.Value,
    fConfidence := fConfidence.Value,
    hrPrev := hrPrev.Value,
    aPerspectiveTransform => perspectiveTransform,
    nNumberOfGoodMatches => numberOfGoodMatches,
    nNumberOfInliers => numberOfInliers);

aPerspectiveTransform.Value := perspectiveTransform;
nNumberOfGoodMatches.Value := numberOfGoodMatches;
nNumberOfInliers.Value := numberOfInliers;
END_METHOD

METHOD PUBLIC PreExecutionCheck
VAR_INPUT
    Check : I_PreExecutionChecks;
END_VAR
Check.IsTrue(ipSrcImage.IsValid, 'ipSrcImage must contain an image');
Check.IsTrue(ipSrcImage.HasChannelCount(1), 'ipSrcImage must have 1 channel');
IF ipSrcImageMask.Value <> 0 THEN
    Check.IsTrue(ipSrcImageMask.IsValid, 'ipSrcImageMask must contain an image when connected');
    Check.IsTrue(IsImage1SizeEqualToImage2Size(ipSrcImage.Value, ipSrcImageMask.Value), 'ipSrcImageMask must have the same size as ipSrcImage');
END_IF
Check.IsTrue(ipRefKeyPoints.IsValid, 'ipRefKeyPoints must contain a container');
Check.IsTrue(ipRefDescriptors.IsValid, 'ipRefDescriptors must contain an image');
Check.IsTrue(nRefImageWidth.Value > 0, 'nRefImageWidth must be greater than 0');
Check.IsTrue(nRefImageHeight.Value > 0, 'nRefImageHeight must be greater than 0');
Check.IsTrue((fMaxDist.Value = -1.0) OR (fMaxDist.Value >= 0.0), 'fMaxDist must be -1 to disable the filter, or at least 0');
Check.IsTrue((fMaxKnnRatio.Value = -1.0) OR
             ((fMaxKnnRatio.Value >= 0.0) AND (fMaxKnnRatio.Value <= 1.0)), 'fMaxKnnRatio must be -1 to disable the filter, or between 0 and 1');
Check.IsTrue((eNormType.Value = ETcVnNormalizationType.TCVN_NT_L1) OR
             (eNormType.Value = ETcVnNormalizationType.TCVN_NT_L2) OR
             (eNormType.Value = ETcVnNormalizationType.TCVN_NT_L2SQR) OR
             (eNormType.Value = ETcVnNormalizationType.TCVN_NT_HAMMING) OR
             (eNormType.Value = ETcVnNormalizationType.TCVN_NT_HAMMING2), 'Unsupported eNormType');
Check.IsTrue((eAlgorithm.Value = ETcVnEstimationAlgorithm.TCVN_EA_DEFAULT) OR
             (eAlgorithm.Value = ETcVnEstimationAlgorithm.TCVN_EA_LMEDS) OR
             (eAlgorithm.Value = ETcVnEstimationAlgorithm.TCVN_EA_RANSAC) OR
             (eAlgorithm.Value = ETcVnEstimationAlgorithm.TCVN_EA_RHO), 'Unsupported eAlgorithm');
// fReprojThreshold is only used by RANSAC and RHO.
Check.IsTrue(((eAlgorithm.Value <> ETcVnEstimationAlgorithm.TCVN_EA_RANSAC) AND
              (eAlgorithm.Value <> ETcVnEstimationAlgorithm.TCVN_EA_RHO)) OR
             (fReprojThreshold.Value > 0.0), 'fReprojThreshold must be greater than 0 for RANSAC and RHO');
Check.IsTrue(nMaxIterations.Value > 0, 'nMaxIterations must be greater than 0');
Check.IsTrue((fConfidence.Value > 0.0) AND (fConfidence.Value < 1.0), 'fConfidence must be between 0 and 1');
END_METHOD

END_FUNCTION_BLOCK

// ---- Nodes/Keypoint Features/Node_F_VN_FindReferenceKeyPointsInImageORB.TcPOU
{attribute 'linkalways'}
{attribute 'no_explicit_call' := 'This FB is a CLASS and must be accessed using methods or properties'}
{attribute 'enable_dynamic_creation'}
FUNCTION_BLOCK Node_F_VN_FindReferenceKeyPointsInImageORB EXTENDS VisionNode
VAR
    ipSrcImage : _ITcVnImage;
    ipRefKeyPoints : _ITcVnContainer;
    ipRefDescriptors : _ITcVnImage;
    nRefImageWidth : _UDINT(0);
    nRefImageHeight : _UDINT(0);
    ipEdgePoints : _ITcVnContainer;
    fMaxDist : _REAL(-1.0);
    fMaxKnnRatio : _REAL(-1.0);
    hrPrev : _HRESULT(S_OK);
    aPerspectiveTransform : _TcVnMatrix3x3_LREAL;
    nNumberOfGoodMatches : _UDINT(0);
    nNumberOfInliers : _UDINT(0);
    hresult : _HRESULT(S_OK);
END_VAR

METHOD PUBLIC Clone : I_Node
VAR
    pNode : POINTER TO Node_F_VN_FindReferenceKeyPointsInImageORB;
END_VAR
pNode := __NEW(Node_F_VN_FindReferenceKeyPointsInImageORB);
Clone := pNode^;
END_METHOD

METHOD FB_init : BOOL
VAR_INPUT
    bInitRetains : BOOL;
    bInCopyCode : BOOL;
END_VAR
AddInput('ipSrcImage', ipSrcImage);
AddInput('ipRefKeyPoints', ipRefKeyPoints);
AddInput('ipRefDescriptors', ipRefDescriptors);
AddInput('nRefImageWidth', nRefImageWidth);
AddInput('nRefImageHeight', nRefImageHeight);
AddOutput('ipEdgePoints', ipEdgePoints);
AddParameter('fMaxDist', fMaxDist);
AddParameter('fMaxKnnRatio', fMaxKnnRatio);
AddInput('hrPrev', hrPrev);
AddOutput('aPerspectiveTransform', aPerspectiveTransform);
AddOutput('nNumberOfGoodMatches', nNumberOfGoodMatches);
AddOutput('nNumberOfInliers', nNumberOfInliers);
AddOutput('hresult', hresult);
END_METHOD

METHOD PROTECTED OnExecute
VAR
    perspectiveTransform : TcVnMatrix3x3_LREAL;
    numberOfGoodMatches : UDINT;
    numberOfInliers : UDINT;
END_VAR
hresult.Value := F_VN_FindReferenceKeyPointsInImageORB(
    ipSrcImage := ipSrcImage.Value,
    ipRefKeyPoints := ipRefKeyPoints.Value,
    ipRefDescriptors := ipRefDescriptors.Value,
    nRefImageWidth := nRefImageWidth.Value,
    nRefImageHeight := nRefImageHeight.Value,
    ipEdgePoints := ipEdgePoints.Value,
    fMaxDist := fMaxDist.Value,
    fMaxKnnRatio := fMaxKnnRatio.Value,
    hrPrev := hrPrev.Value,
    aPerspectiveTransform => perspectiveTransform,
    nNumberOfGoodMatches => numberOfGoodMatches,
    nNumberOfInliers => numberOfInliers);

aPerspectiveTransform.Value := perspectiveTransform;
nNumberOfGoodMatches.Value := numberOfGoodMatches;
nNumberOfInliers.Value := numberOfInliers;
END_METHOD

METHOD PUBLIC PreExecutionCheck
VAR_INPUT
    Check : I_PreExecutionChecks;
END_VAR
Check.IsTrue(ipSrcImage.IsValid, 'ipSrcImage must contain an image');
Check.IsTrue(ipSrcImage.HasChannelCount(1), 'ipSrcImage must have 1 channel');
Check.IsTrue(ipRefKeyPoints.IsValid, 'ipRefKeyPoints must contain a container');
Check.IsTrue(ipRefDescriptors.IsValid, 'ipRefDescriptors must contain an image');
Check.IsTrue(nRefImageWidth.Value > 0, 'nRefImageWidth must be greater than 0');
Check.IsTrue(nRefImageHeight.Value > 0, 'nRefImageHeight must be greater than 0');
Check.IsTrue((fMaxDist.Value = -1.0) OR (fMaxDist.Value >= 0.0), 'fMaxDist must be -1 to disable the filter, or at least 0');
Check.IsTrue((fMaxKnnRatio.Value = -1.0) OR
             ((fMaxKnnRatio.Value >= 0.0) AND (fMaxKnnRatio.Value <= 1.0)), 'fMaxKnnRatio must be -1 to disable the filter, or between 0 and 1');
END_METHOD

END_FUNCTION_BLOCK

// ---- Nodes/Keypoint Features/Node_F_VN_FindReferenceKeyPointsInImageORBExp.TcPOU
{attribute 'linkalways'}
{attribute 'no_explicit_call' := 'This FB is a CLASS and must be accessed using methods or properties'}
{attribute 'enable_dynamic_creation'}
FUNCTION_BLOCK Node_F_VN_FindReferenceKeyPointsInImageORBExp EXTENDS VisionNode
VAR
    ipSrcImage : _ITcVnImage;
    ipRefKeyPoints : _ITcVnContainer;
    ipRefDescriptors : _ITcVnImage;
    nRefImageWidth : _UDINT(0);
    nRefImageHeight : _UDINT(0);
    ipEdgePoints : _ITcVnContainer;
    fMaxDist : _REAL(-1.0);
    fMaxKnnRatio : _REAL(-1.0);
    eNormType : _ETcVnNormalizationType(ETcVnNormalizationType.TCVN_NT_HAMMING);
    ipSrcImageMask : _ITcVnImage;
    stOrbParams : _TcVnParamsORB;
    eAlgorithm : _ETcVnEstimationAlgorithm(ETcVnEstimationAlgorithm.TCVN_EA_RANSAC);
    fReprojThreshold : _LREAL(3.0);
    nMaxIterations : _UDINT(2000);
    fConfidence : _LREAL(0.995);
    hrPrev : _HRESULT(S_OK);
    aPerspectiveTransform : _TcVnMatrix3x3_LREAL;
    nNumberOfGoodMatches : _UDINT(0);
    nNumberOfInliers : _UDINT(0);
    hresult : _HRESULT(S_OK);
END_VAR

METHOD PUBLIC Clone : I_Node
VAR
    pNode : POINTER TO Node_F_VN_FindReferenceKeyPointsInImageORBExp;
END_VAR
pNode := __NEW(Node_F_VN_FindReferenceKeyPointsInImageORBExp);
Clone := pNode^;
END_METHOD

METHOD FB_init : BOOL
VAR_INPUT
    bInitRetains : BOOL;
    bInCopyCode : BOOL;
END_VAR
AddInput('ipSrcImage', ipSrcImage);
AddInput('ipRefKeyPoints', ipRefKeyPoints);
AddInput('ipRefDescriptors', ipRefDescriptors);
AddInput('nRefImageWidth', nRefImageWidth);
AddInput('nRefImageHeight', nRefImageHeight);
AddOutput('ipEdgePoints', ipEdgePoints);
AddParameter('fMaxDist', fMaxDist);
AddParameter('fMaxKnnRatio', fMaxKnnRatio);
AddParameter('eNormType', eNormType);
AddInput('ipSrcImageMask', ipSrcImageMask);
AddInput('stOrbParams', stOrbParams);
AddParameter('eAlgorithm', eAlgorithm);
AddParameter('fReprojThreshold', fReprojThreshold);
AddParameter('nMaxIterations', nMaxIterations);
AddParameter('fConfidence', fConfidence);
AddInput('hrPrev', hrPrev);
AddOutput('aPerspectiveTransform', aPerspectiveTransform);
AddOutput('nNumberOfGoodMatches', nNumberOfGoodMatches);
AddOutput('nNumberOfInliers', nNumberOfInliers);
AddOutput('hresult', hresult);
END_METHOD

METHOD PROTECTED OnExecute
VAR
    perspectiveTransform : TcVnMatrix3x3_LREAL;
    numberOfGoodMatches : UDINT;
    numberOfInliers : UDINT;
END_VAR
hresult.Value := F_VN_FindReferenceKeyPointsInImageORBExp(
    ipSrcImage := ipSrcImage.Value,
    ipRefKeyPoints := ipRefKeyPoints.Value,
    ipRefDescriptors := ipRefDescriptors.Value,
    nRefImageWidth := nRefImageWidth.Value,
    nRefImageHeight := nRefImageHeight.Value,
    ipEdgePoints := ipEdgePoints.Value,
    fMaxDist := fMaxDist.Value,
    fMaxKnnRatio := fMaxKnnRatio.Value,
    eNormType := eNormType.Value,
    ipSrcImageMask := ipSrcImageMask.Value,
    stOrbParams := stOrbParams.Value,
    eAlgorithm := eAlgorithm.Value,
    fReprojThreshold := fReprojThreshold.Value,
    nMaxIterations := nMaxIterations.Value,
    fConfidence := fConfidence.Value,
    hrPrev := hrPrev.Value,
    aPerspectiveTransform => perspectiveTransform,
    nNumberOfGoodMatches => numberOfGoodMatches,
    nNumberOfInliers => numberOfInliers);

aPerspectiveTransform.Value := perspectiveTransform;
nNumberOfGoodMatches.Value := numberOfGoodMatches;
nNumberOfInliers.Value := numberOfInliers;
END_METHOD

METHOD PUBLIC PreExecutionCheck
VAR_INPUT
    Check : I_PreExecutionChecks;
END_VAR
Check.IsTrue(ipSrcImage.IsValid, 'ipSrcImage must contain an image');
Check.IsTrue(ipSrcImage.HasChannelCount(1), 'ipSrcImage must have 1 channel');
IF ipSrcImageMask.Value <> 0 THEN
    Check.IsTrue(ipSrcImageMask.IsValid, 'ipSrcImageMask must contain an image when connected');
    Check.IsTrue(IsImage1SizeEqualToImage2Size(ipSrcImage.Value, ipSrcImageMask.Value), 'ipSrcImageMask must have the same size as ipSrcImage');
END_IF
Check.IsTrue(ipRefKeyPoints.IsValid, 'ipRefKeyPoints must contain a container');
Check.IsTrue(ipRefDescriptors.IsValid, 'ipRefDescriptors must contain an image');
Check.IsTrue(nRefImageWidth.Value > 0, 'nRefImageWidth must be greater than 0');
Check.IsTrue(nRefImageHeight.Value > 0, 'nRefImageHeight must be greater than 0');
Check.IsTrue((fMaxDist.Value = -1.0) OR (fMaxDist.Value >= 0.0), 'fMaxDist must be -1 to disable the filter, or at least 0');
Check.IsTrue((fMaxKnnRatio.Value = -1.0) OR
             ((fMaxKnnRatio.Value >= 0.0) AND (fMaxKnnRatio.Value <= 1.0)), 'fMaxKnnRatio must be -1 to disable the filter, or between 0 and 1');
Check.IsTrue((eNormType.Value = ETcVnNormalizationType.TCVN_NT_L1) OR
             (eNormType.Value = ETcVnNormalizationType.TCVN_NT_L2) OR
             (eNormType.Value = ETcVnNormalizationType.TCVN_NT_L2SQR) OR
             (eNormType.Value = ETcVnNormalizationType.TCVN_NT_HAMMING) OR
             (eNormType.Value = ETcVnNormalizationType.TCVN_NT_HAMMING2), 'Unsupported eNormType');
Check.IsTrue(stOrbParams.Value.fPyramidScale > 1, 'fPyramidScale must be greater than 1');
Check.IsTrue(stOrbParams.Value.nFirstLevel = 0, 'nFirstLevel must be equal to 0');
Check.IsTrue((stOrbParams.Value.nBriefPoints >= 2) AND (stOrbParams.Value.nBriefPoints <= 4), 'nBriefPoints must be between 2 and 4');
Check.IsTrue((eAlgorithm.Value = ETcVnEstimationAlgorithm.TCVN_EA_DEFAULT) OR
             (eAlgorithm.Value = ETcVnEstimationAlgorithm.TCVN_EA_LMEDS) OR
             (eAlgorithm.Value = ETcVnEstimationAlgorithm.TCVN_EA_RANSAC) OR
             (eAlgorithm.Value = ETcVnEstimationAlgorithm.TCVN_EA_RHO), 'Unsupported eAlgorithm');
// fReprojThreshold is only used by RANSAC and RHO.
Check.IsTrue(((eAlgorithm.Value <> ETcVnEstimationAlgorithm.TCVN_EA_RANSAC) AND
              (eAlgorithm.Value <> ETcVnEstimationAlgorithm.TCVN_EA_RHO)) OR
             (fReprojThreshold.Value > 0.0), 'fReprojThreshold must be greater than 0 for RANSAC and RHO');
Check.IsTrue(nMaxIterations.Value > 0, 'nMaxIterations must be greater than 0');
Check.IsTrue((fConfidence.Value > 0.0) AND (fConfidence.Value < 1.0), 'fConfidence must be between 0 and 1');
END_METHOD

END_FUNCTION_BLOCK

// ---- Nodes/Keypoint Features/Node_F_VN_KeyPointsAGAST.TcPOU
{attribute 'linkalways'} 
{attribute 'no_explicit_call' := 'This FB is a CLASS and must be accessed using methods or properties'}
{attribute 'enable_dynamic_creation'}
FUNCTION_BLOCK Node_F_VN_KeyPointsAGAST EXTENDS VisionNode
VAR
    ipSrcImage : _ITcVnImage;
    ipKeyPoints : _ITcVnContainer;
    hrPrev : _HRESULT(S_OK);
	hresult : _HRESULT(S_OK);
END_VAR

METHOD PUBLIC  Clone : I_Node
VAR
	pNode : POINTER TO Node_F_VN_KeyPointsAGAST;
END_VAR
pNode := __NEW(Node_F_VN_KeyPointsAGAST);
Clone := pNode^;
END_METHOD

METHOD FB_init : BOOL
VAR_INPUT
	bInitRetains : BOOL; // if TRUE, the retain variables are initialized (warm start / cold start)
	bInCopyCode : BOOL;  // if TRUE, the instance afterwards gets moved into the copy code (online change)
END_VAR
AddInput('ipSrcImage', ipSrcImage);
AddInput('hrPrev', hrPrev);
AddOutput('ipKeyPoints', ipKeyPoints);
AddOutput('hresult',hresult);
END_METHOD

METHOD PROTECTED OnExecute
hresult.Value := F_VN_KeyPointsAGAST(
	ipSrcImage := ipSrcImage.Value,
    ipKeyPoints := ipKeyPoints.Value,
	hrPrev:= hrPrev.Value);
END_METHOD

METHOD PUBLIC PreExecutionCheck
VAR_INPUT
	Check : I_PreExecutionChecks;
END_VAR
Check.IsTrue(ipSrcImage.IsValid, 'ipSrcImage must contain an image');
Check.IsTrue(ipSrcImage.HasChannelCount(1), 'ipSrcImage must have 1 channel');
END_METHOD

END_FUNCTION_BLOCK

// ---- Nodes/Keypoint Features/Node_F_VN_KeyPointsAGASTExp.TcPOU
{attribute 'linkalways'} 
{attribute 'no_explicit_call' := 'This FB is a CLASS and must be accessed using methods or properties'}
{attribute 'enable_dynamic_creation'}
FUNCTION_BLOCK Node_F_VN_KeyPointsAGASTExp EXTENDS VisionNode
VAR
    ipSrcImage : _ITcVnImage;
    ipKeyPoints : _ITcVnContainer;
    ipMask : _ITcVnImage;
    stParams : _TcVnParamsAGAST;
    hrPrev : _HRESULT(S_OK);
	hresult : _HRESULT(S_OK);
END_VAR

METHOD PUBLIC  Clone : I_Node
VAR
	pNode : POINTER TO Node_F_VN_KeyPointsAGASTExp;
END_VAR
pNode := __NEW(Node_F_VN_KeyPointsAGASTExp);
Clone := pNode^;
END_METHOD

METHOD FB_init : BOOL
VAR_INPUT
	bInitRetains : BOOL; // if TRUE, the retain variables are initialized (warm start / cold start)
	bInCopyCode : BOOL;  // if TRUE, the instance afterwards gets moved into the copy code (online change)
END_VAR
AddInput('ipSrcImage', ipSrcImage);
AddInput('ipMask', ipMask);
AddInput('stParams', stParams);
AddInput('hrPrev', hrPrev);
AddOutput('ipKeyPoints', ipKeyPoints);
AddOutput('hresult',hresult);
END_METHOD

METHOD PROTECTED OnExecute
hresult.Value := F_VN_KeyPointsAGASTExp(
	ipSrcImage := ipSrcImage.Value,
    ipKeyPoints := ipKeyPoints.Value,
    ipMask := ipMask.Value,
    stParams := stParams.Value,
	hrPrev:= hrPrev.Value);
END_METHOD

METHOD PUBLIC PreExecutionCheck
VAR_INPUT
	Check : I_PreExecutionChecks;
END_VAR
Check.IsTrue(ipSrcImage.IsValid, 'ipSrcImage must contain an image');
Check.IsTrue(ipSrcImage.HasChannelCount(1), 'ipSrcImage must have 1 channel');
END_METHOD

END_FUNCTION_BLOCK

// ---- Nodes/Keypoint Features/Node_F_VN_GetMatchCoordinates.TcPOU
{attribute 'linkalways'} 
{attribute 'no_explicit_call' := 'This FB is a CLASS and must be accessed using methods or properties'}
{attribute 'enable_dynamic_creation'}
FUNCTION_BLOCK Node_F_VN_GetMatchCoordinates EXTENDS VisionNode
VAR
    ipQueryKeyPoints : _ITcVnContainer;
    ipTrainKeyPoints : _ITcVnContainer;
    ipMatches : _ITcVnContainer;
    ipQueryCoordinates : _ITcVnContainer;
    ipTrainCoordinates : _ITcVnContainer;
    hrPrev : _HRESULT(S_OK);
	hresult : _HRESULT(S_OK);
END_VAR

METHOD PUBLIC  Clone : I_Node
VAR
	pNode : POINTER TO Node_F_VN_GetMatchCoordinates;
END_VAR
pNode := __NEW(Node_F_VN_GetMatchCoordinates);
Clone := pNode^;
END_METHOD

METHOD FB_init : BOOL
VAR_INPUT
	bInitRetains : BOOL; // if TRUE, the retain variables are initialized (warm start / cold start)
	bInCopyCode : BOOL;  // if TRUE, the instance afterwards gets moved into the copy code (online change)
END_VAR
AddInput('ipQueryKeyPoints', ipQueryKeyPoints);
AddInput('ipTrainKeyPoints', ipTrainKeyPoints);
AddInput('ipMatches', ipMatches);
AddInput('hrPrev', hrPrev);
AddOutput('ipQueryCoordinates', ipQueryCoordinates);
AddOutput('ipTrainCoordinates', ipTrainCoordinates);
AddOutput('hresult',hresult);
END_METHOD

METHOD PROTECTED OnExecute
hresult.Value := F_VN_GetMatchCoordinates(
	ipQueryKeyPoints := ipQueryKeyPoints.Value,
    ipTrainKeyPoints := ipTrainKeyPoints.Value,
    ipMatches := ipMatches.Value,
    ipQueryCoordinates := ipQueryCoordinates.Value,
    ipTrainCoordinates := ipTrainCoordinates.Value,
	hrPrev:= hrPrev.Value);
END_METHOD

METHOD PUBLIC PreExecutionCheck
VAR_INPUT
	Check : I_PreExecutionChecks;
END_VAR
Check.IsTrue(ipQueryKeyPoints.IsValid, 'ipQueryKeyPoints must be a valid container');
Check.IsTrue(ipQueryKeyPoints.IsType(TC_GLOBAL_CONST_LIST.ContainerType_Vector_TcVnKeyPoint), 'ipQueryKeyPoints contains incorrect type');

Check.IsTrue(ipTrainKeyPoints.IsValid, 'ipTrainKeyPoints must be a valid container');
Check.IsTrue(ipTrainKeyPoints.IsType(TC_GLOBAL_CONST_LIST.ContainerType_Vector_TcVnKeyPoint), 'ipTrainKeyPoints contains incorrect type');

Check.IsTrue(ipMatches.IsValid, 'ipMatches must be a valid container');
Check.IsTrue(ipMatches.IsType(TC_GLOBAL_CONST_LIST.ContainerType_Vector_TcVnDMatch), 'ipMatches contains incorrect type');
END_METHOD

END_FUNCTION_BLOCK

// ---- Nodes/Keypoint Features/Node_F_VN_KeyPointsAndDescriptorsAKAZE.TcPOU
{attribute 'linkalways'} 
{attribute 'no_explicit_call' := 'This FB is a CLASS and must be accessed using methods or properties'}
{attribute 'enable_dynamic_creation'}
FUNCTION_BLOCK Node_F_VN_KeyPointsAndDescriptorsAKAZE EXTENDS VisionNode
VAR
    ipSrcImage : _ITcVnImage;
    ipKeyPoints : _ITcVnContainer;
    ipDescriptors : _ITcVnImage;
    hrPrev : _HRESULT(S_OK);
	hresult : _HRESULT(S_OK);
END_VAR

METHOD PUBLIC  Clone : I_Node
VAR
	pNode : POINTER TO Node_F_VN_KeyPointsAndDescriptorsAKAZE;
END_VAR
pNode := __NEW(Node_F_VN_KeyPointsAndDescriptorsAKAZE);
Clone := pNode^;
END_METHOD

METHOD FB_init : BOOL
VAR_INPUT
	bInitRetains : BOOL; // if TRUE, the retain variables are initialized (warm start / cold start)
	bInCopyCode : BOOL;  // if TRUE, the instance afterwards gets moved into the copy code (online change)
END_VAR
AddInput('ipSrcImage', ipSrcImage);
AddInput('hrPrev', hrPrev);
AddOutput('ipKeyPoints', ipKeyPoints);
AddOutput('ipDescriptors', ipDescriptors);
AddOutput('hresult',hresult);
END_METHOD

METHOD PROTECTED OnExecute
hresult.Value := F_VN_KeyPointsAndDescriptorsAKAZE(
	ipSrcImage := ipSrcImage.Value,
    ipKeyPoints := ipKeyPoints.Value,
    ipDescriptors := ipDescriptors.Value,
	hrPrev:= hrPrev.Value);
END_METHOD

METHOD PUBLIC PreExecutionCheck
VAR_INPUT
	Check : I_PreExecutionChecks;
END_VAR
Check.IsTrue(ipSrcImage.IsValid, 'ipSrcImage must contain an image');
Check.IsTrue(ipSrcImage.HasChannelCount(1), 'ipSrcImage must have 1 channel');
END_METHOD

END_FUNCTION_BLOCK

// ---- Nodes/Keypoint Features/Node_F_VN_KeyPointsAndDescriptorsAKAZEExp.TcPOU
{attribute 'linkalways'} 
{attribute 'no_explicit_call' := 'This FB is a CLASS and must be accessed using methods or properties'}
{attribute 'enable_dynamic_creation'}
FUNCTION_BLOCK Node_F_VN_KeyPointsAndDescriptorsAKAZEExp EXTENDS VisionNode
VAR
    ipSrcImage : _ITcVnImage;
    ipKeyPoints : _ITcVnContainer;
    ipDescriptors : _ITcVnImage;
    ipMask : _ITcVnImage;
    stParams : _TcVnParamsAKAZE;
    hrPrev : _HRESULT(S_OK);
	hresult : _HRESULT(S_OK);
END_VAR

METHOD PUBLIC  Clone : I_Node
VAR
	pNode : POINTER TO Node_F_VN_KeyPointsAndDescriptorsAKAZEExp;
END_VAR
pNode := __NEW(Node_F_VN_KeyPointsAndDescriptorsAKAZEExp);
Clone := pNode^;
END_METHOD

METHOD FB_init : BOOL
VAR_INPUT
	bInitRetains : BOOL; // if TRUE, the retain variables are initialized (warm start / cold start)
	bInCopyCode : BOOL;  // if TRUE, the instance afterwards gets moved into the copy code (online change)
END_VAR
AddInput('ipSrcImage', ipSrcImage);
AddInput('ipMask', ipMask);
AddInput('stParams', stParams);
AddInput('hrPrev', hrPrev);
AddOutput('ipKeyPoints', ipKeyPoints);
AddOutput('ipDescriptors', ipDescriptors);
AddOutput('hresult',hresult);
END_METHOD

METHOD PROTECTED OnExecute
hresult.Value := F_VN_KeyPointsAndDescriptorsAKAZEExp(
	ipSrcImage := ipSrcImage.Value,
    ipKeyPoints := ipKeyPoints.Value,
    ipDescriptors := ipDescriptors.Value,
    ipMask := ipMask.Value,
    stParams := stParams.Value,
	hrPrev:= hrPrev.Value);
END_METHOD

METHOD PUBLIC PreExecutionCheck
VAR_INPUT
	Check : I_PreExecutionChecks;
END_VAR
Check.IsTrue(ipSrcImage.IsValid, 'ipSrcImage must contain an image');
Check.IsTrue(ipSrcImage.HasChannelCount(1), 'ipSrcImage must have 1 channel');

IF ((stParams.Value.eDescrType = ETcVnFeatureDescriptorTypeAKAZE.TCVN_FDT_AKAZE_MLDB) OR 
    (stParams.Value.eDescrType = ETcVnFeatureDescriptorTypeAKAZE.TCVN_FDT_AKAZE_MLDB_UPRIGHT)) THEN
    Check.IsTrue(stParams.Value.nDescrChannels = 3, 'nDescrChannels must be 3 when using AKAZE_MLDB');
END_IF
END_METHOD

END_FUNCTION_BLOCK

// ---- Nodes/Keypoint Features/Node_F_VN_KeyPointsAndDescriptorsBRISKExp.TcPOU
{attribute 'linkalways'} 
{attribute 'no_explicit_call' := 'This FB is a CLASS and must be accessed using methods or properties'}
{attribute 'enable_dynamic_creation'}
FUNCTION_BLOCK Node_F_VN_KeyPointsAndDescriptorsBRISKExp EXTENDS VisionNode
VAR
    ipSrcImage : _ITcVnImage;
    ipKeyPoints : _ITcVnContainer;
    ipDescriptors : _ITcVnImage;
    ipMask : _ITcVnImage;
    stParams : _TcVnParamsBRISK;
    hrPrev : _HRESULT(S_OK);
	hresult : _HRESULT(S_OK);
END_VAR

METHOD PUBLIC  Clone : I_Node
VAR
	pNode : POINTER TO Node_F_VN_KeyPointsAndDescriptorsBRISKExp;
END_VAR
pNode := __NEW(Node_F_VN_KeyPointsAndDescriptorsBRISKExp);
Clone := pNode^;
END_METHOD

METHOD FB_init : BOOL
VAR_INPUT
	bInitRetains : BOOL; // if TRUE, the retain variables are initialized (warm start / cold start)
	bInCopyCode : BOOL;  // if TRUE, the instance afterwards gets moved into the copy code (online change)
END_VAR
AddInput('ipSrcImage', ipSrcImage);
AddInput('ipMask', ipMask);
AddInput('stParams', stParams);
AddInput('hrPrev', hrPrev);
AddOutput('ipKeyPoints', ipKeyPoints);
AddOutput('ipDescriptors', ipDescriptors);
AddOutput('hresult',hresult);
END_METHOD

METHOD PROTECTED OnExecute
hresult.Value := F_VN_KeyPointsAndDescriptorsBRISKExp(
	ipSrcImage := ipSrcImage.Value,
    ipKeyPoints := ipKeyPoints.Value,
    ipDescriptors := ipDescriptors.Value,
    ipMask := ipMask.Value,
    stParams := stParams.Value,
	hrPrev:= hrPrev.Value);
END_METHOD

METHOD PUBLIC PreExecutionCheck
VAR_INPUT
	Check : I_PreExecutionChecks;
END_VAR
Check.IsTrue(ipSrcImage.IsValid, 'ipSrcImage must contain an image');
Check.IsTrue(ipSrcImage.HasChannelCount(1), 'ipSrcImage must have 1 channel');
END_METHOD

END_FUNCTION_BLOCK

// ---- Nodes/Keypoint Features/Node_F_VN_KeyPointsAndDescriptorsBRISK.TcPOU
{attribute 'linkalways'} 
{attribute 'no_explicit_call' := 'This FB is a CLASS and must be accessed using methods or properties'}
{attribute 'enable_dynamic_creation'}
FUNCTION_BLOCK Node_F_VN_KeyPointsAndDescriptorsBRISK EXTENDS VisionNode
VAR
    ipSrcImage : _ITcVnImage;
    ipKeyPoints : _ITcVnContainer;
    ipDescriptors : _ITcVnImage;
    hrPrev : _HRESULT(S_OK);
	hresult : _HRESULT(S_OK);
END_VAR

METHOD PUBLIC  Clone : I_Node
VAR
	pNode : POINTER TO Node_F_VN_KeyPointsAndDescriptorsBRISK;
END_VAR
pNode := __NEW(Node_F_VN_KeyPointsAndDescriptorsBRISK);
Clone := pNode^;
END_METHOD

METHOD FB_init : BOOL
VAR_INPUT
	bInitRetains : BOOL; // if TRUE, the retain variables are initialized (warm start / cold start)
	bInCopyCode : BOOL;  // if TRUE, the instance afterwards gets moved into the copy code (online change)
END_VAR
AddInput('ipSrcImage', ipSrcImage);
AddInput('hrPrev', hrPrev);
AddOutput('ipKeyPoints', ipKeyPoints);
AddOutput('ipDescriptors', ipDescriptors);
AddOutput('hresult',hresult);
END_METHOD

METHOD PROTECTED OnExecute
hresult.Value := F_VN_KeyPointsAndDescriptorsBRISK(
	ipSrcImage := ipSrcImage.Value,
    ipKeyPoints := ipKeyPoints.Value,
    ipDescriptors := ipDescriptors.Value,
	hrPrev:= hrPrev.Value);
END_METHOD

METHOD PUBLIC PreExecutionCheck
VAR_INPUT
	Check : I_PreExecutionChecks;
END_VAR
Check.IsTrue(ipSrcImage.IsValid, 'ipSrcImage must contain an image');
Check.IsTrue(ipSrcImage.HasChannelCount(1), 'ipSrcImage must have 1 channel');
END_METHOD

END_FUNCTION_BLOCK

// ---- Nodes/Keypoint Features/Node_F_VN_KeyPointsAndDescriptorsKAZEExp.TcPOU
{attribute 'linkalways'} 
{attribute 'no_explicit_call' := 'This FB is a CLASS and must be accessed using methods or properties'}
{attribute 'enable_dynamic_creation'}
FUNCTION_BLOCK Node_F_VN_KeyPointsAndDescriptorsKAZEExp EXTENDS VisionNode
VAR
    ipSrcImage : _ITcVnImage;
    ipKeyPoints : _ITcVnContainer;
    ipDescriptors : _ITcVnImage;
    ipMask : _ITcVnImage;
    stParams : _TcVnParamsKAZE;
    hrPrev : _HRESULT(S_OK);
	hresult : _HRESULT(S_OK);
END_VAR

METHOD PUBLIC  Clone : I_Node
VAR
	pNode : POINTER TO Node_F_VN_KeyPointsAndDescriptorsKAZEExp;
END_VAR
pNode := __NEW(Node_F_VN_KeyPointsAndDescriptorsKAZEExp);
Clone := pNode^;
END_METHOD

METHOD FB_init : BOOL
VAR_INPUT
	bInitRetains : BOOL; // if TRUE, the retain variables are initialized (warm start / cold start)
	bInCopyCode : BOOL;  // if TRUE, the instance afterwards gets moved into the copy code (online change)
END_VAR
AddInput('ipSrcImage', ipSrcImage);
AddInput('ipMask', ipMask);
AddInput('stParams', stParams);
AddInput('hrPrev', hrPrev);
AddOutput('ipKeyPoints', ipKeyPoints);
AddOutput('ipDescriptors', ipDescriptors);
AddOutput('hresult',hresult);
END_METHOD

METHOD PROTECTED OnExecute
hresult.Value := F_VN_KeyPointsAndDescriptorsKAZEExp(
	ipSrcImage := ipSrcImage.Value,
    ipKeyPoints := ipKeyPoints.Value,
    ipDescriptors := ipDescriptors.Value,
    ipMask := ipMask.Value,
    stParams := stParams.Value,
	hrPrev:= hrPrev.Value);
END_METHOD

METHOD PUBLIC PreExecutionCheck
VAR_INPUT
	Check : I_PreExecutionChecks;
END_VAR
Check.IsTrue(ipSrcImage.IsValid, 'ipSrcImage must contain an image');
Check.IsTrue(ipSrcImage.HasChannelCount(1), 'ipSrcImage must have 1 channel');
END_METHOD

END_FUNCTION_BLOCK

// ---- Nodes/Keypoint Features/Node_F_VN_KeyPointsAndDescriptorsKAZE.TcPOU
{attribute 'linkalways'} 
{attribute 'no_explicit_call' := 'This FB is a CLASS and must be accessed using methods or properties'}
{attribute 'enable_dynamic_creation'}
FUNCTION_BLOCK Node_F_VN_KeyPointsAndDescriptorsKAZE EXTENDS VisionNode
VAR
    ipSrcImage : _ITcVnImage;
    ipKeyPoints : _ITcVnContainer;
    ipDescriptors : _ITcVnImage;
    hrPrev : _HRESULT(S_OK);
	hresult : _HRESULT(S_OK);
END_VAR

METHOD PUBLIC  Clone : I_Node
VAR
	pNode : POINTER TO Node_F_VN_KeyPointsAndDescriptorsKAZE;
END_VAR
pNode := __NEW(Node_F_VN_KeyPointsAndDescriptorsKAZE);
Clone := pNode^;
END_METHOD

METHOD FB_init : BOOL
VAR_INPUT
	bInitRetains : BOOL; // if TRUE, the retain variables are initialized (warm start / cold start)
	bInCopyCode : BOOL;  // if TRUE, the instance afterwards gets moved into the copy code (online change)
END_VAR
AddInput('ipSrcImage', ipSrcImage);
AddInput('hrPrev', hrPrev);
AddOutput('ipKeyPoints', ipKeyPoints);
AddOutput('ipDescriptors', ipDescriptors);
AddOutput('hresult',hresult);
END_METHOD

METHOD PROTECTED OnExecute
hresult.Value := F_VN_KeyPointsAndDescriptorsKAZE(
	ipSrcImage := ipSrcImage.Value,
    ipKeyPoints := ipKeyPoints.Value,
    ipDescriptors := ipDescriptors.Value,
	hrPrev:= hrPrev.Value);
END_METHOD

METHOD PUBLIC PreExecutionCheck
VAR_INPUT
	Check : I_PreExecutionChecks;
END_VAR
Check.IsTrue(ipSrcImage.IsValid, 'ipSrcImage must contain an image');
Check.IsTrue(ipSrcImage.HasChannelCount(1), 'ipSrcImage must have 1 channel');
END_METHOD

END_FUNCTION_BLOCK

// ---- Nodes/Keypoint Features/Node_F_VN_KeyPointsAndDescriptorsORBExp.TcPOU
{attribute 'linkalways'} 
{attribute 'no_explicit_call' := 'This FB is a CLASS and must be accessed using methods or properties'}
{attribute 'enable_dynamic_creation'}
FUNCTION_BLOCK Node_F_VN_KeyPointsAndDescriptorsORBExp EXTENDS VisionNode
VAR
    ipSrcImage : _ITcVnImage;
    ipKeyPoints : _ITcVnContainer;
    ipDescriptors : _ITcVnImage;
    ipMask : _ITcVnImage;
    stParams : _TcVnParamsORB;
    hrPrev : _HRESULT(S_OK);
	hresult : _HRESULT(S_OK);
END_VAR

METHOD PUBLIC  Clone : I_Node
VAR
	pNode : POINTER TO Node_F_VN_KeyPointsAndDescriptorsORBExp;
END_VAR
pNode := __NEW(Node_F_VN_KeyPointsAndDescriptorsORBExp);
Clone := pNode^;
END_METHOD

METHOD FB_init : BOOL
VAR_INPUT
	bInitRetains : BOOL; // if TRUE, the retain variables are initialized (warm start / cold start)
	bInCopyCode : BOOL;  // if TRUE, the instance afterwards gets moved into the copy code (online change)
END_VAR
AddInput('ipSrcImage', ipSrcImage);
AddInput('ipMask', ipMask);
AddInput('stParams', stParams);
AddInput('hrPrev', hrPrev);
AddOutput('ipKeyPoints', ipKeyPoints);
AddOutput('ipDescriptors', ipDescriptors);
AddOutput('hresult',hresult);
END_METHOD

METHOD PROTECTED OnExecute
hresult.Value := F_VN_KeyPointsAndDescriptorsORBExp(
	ipSrcImage := ipSrcImage.Value,
    ipKeyPoints := ipKeyPoints.Value,
    ipDescriptors := ipDescriptors.Value,
    ipMask := ipMask.Value,
    stParams := stParams.Value,
	hrPrev:= hrPrev.Value);
END_METHOD

METHOD PUBLIC PreExecutionCheck
VAR_INPUT
	Check : I_PreExecutionChecks;
END_VAR
Check.IsTrue(ipSrcImage.IsValid, 'ipSrcImage must contain an image');
Check.IsTrue(ipSrcImage.HasChannelCount(1), 'ipSrcImage must have 1 channel');
Check.IsTrue(stParams.Value.fPyramidScale > 1, 'fPyramidScale must be greater than 1');
Check.IsTrue(stParams.Value.nFirstLevel = 0, 'nFirstLevel must be equal to 0');
Check.IsTrue((stParams.Value.nBriefPoints >= 2) AND (stParams.Value.nBriefPoints <= 4), 'nBriefPoints must be between 2 and 4');
END_METHOD

END_FUNCTION_BLOCK

// ---- Nodes/Keypoint Features/Node_F_VN_KeyPointsAndDescriptorsORB.TcPOU
{attribute 'linkalways'} 
{attribute 'no_explicit_call' := 'This FB is a CLASS and must be accessed using methods or properties'}
{attribute 'enable_dynamic_creation'}
FUNCTION_BLOCK Node_F_VN_KeyPointsAndDescriptorsORB EXTENDS VisionNode
VAR
    ipSrcImage : _ITcVnImage;
    ipKeyPoints : _ITcVnContainer;
    ipDescriptors : _ITcVnImage;
    hrPrev : _HRESULT(S_OK);
	hresult : _HRESULT(S_OK);
END_VAR

METHOD PUBLIC  Clone : I_Node
VAR
	pNode : POINTER TO Node_F_VN_KeyPointsAndDescriptorsORB;
END_VAR
pNode := __NEW(Node_F_VN_KeyPointsAndDescriptorsORB);
Clone := pNode^;
END_METHOD

METHOD FB_init : BOOL
VAR_INPUT
	bInitRetains : BOOL; // if TRUE, the retain variables are initialized (warm start / cold start)
	bInCopyCode : BOOL;  // if TRUE, the instance afterwards gets moved into the copy code (online change)
END_VAR
AddInput('ipSrcImage', ipSrcImage);
AddInput('hrPrev', hrPrev);
AddOutput('ipKeyPoints', ipKeyPoints);
AddOutput('ipDescriptors', ipDescriptors);
AddOutput('hresult',hresult);
END_METHOD

METHOD PROTECTED OnExecute
hresult.Value := F_VN_KeyPointsAndDescriptorsORB(
	ipSrcImage := ipSrcImage.Value,
    ipKeyPoints := ipKeyPoints.Value,
    ipDescriptors := ipDescriptors.Value,
	hrPrev:= hrPrev.Value);
END_METHOD

METHOD PUBLIC PreExecutionCheck
VAR_INPUT
	Check : I_PreExecutionChecks;
END_VAR
Check.IsTrue(ipSrcImage.IsValid, 'ipSrcImage must contain an image');
Check.IsTrue(ipSrcImage.HasChannelCount(1), 'ipSrcImage must have 1 channel');
END_METHOD

END_FUNCTION_BLOCK

// ---- Nodes/Keypoint Features/Node_F_VN_KeyPointsFASTExp.TcPOU
{attribute 'linkalways'} 
{attribute 'no_explicit_call' := 'This FB is a CLASS and must be accessed using methods or properties'}
{attribute 'enable_dynamic_creation'}
FUNCTION_BLOCK Node_F_VN_KeyPointsFASTExp EXTENDS VisionNode
VAR
    ipSrcImage : _ITcVnImage;
    ipKeyPoints : _ITcVnContainer;
    ipMask : _ITcVnImage;
    stParams : _TcVnParamsFAST;
    hrPrev : _HRESULT(S_OK);
	hresult : _HRESULT(S_OK);
END_VAR

METHOD PUBLIC  Clone : I_Node
VAR
	pNode : POINTER TO Node_F_VN_KeyPointsFASTExp;
END_VAR
pNode := __NEW(Node_F_VN_KeyPointsFASTExp);
Clone := pNode^;
END_METHOD

METHOD FB_init : BOOL
VAR_INPUT
	bInitRetains : BOOL; // if TRUE, the retain variables are initialized (warm start / cold start)
	bInCopyCode : BOOL;  // if TRUE, the instance afterwards gets moved into the copy code (online change)
END_VAR
AddInput('ipSrcImage', ipSrcImage);
AddInput('ipMask', ipMask);
AddInput('stParams', stParams);
AddInput('hrPrev', hrPrev);
AddOutput('ipKeyPoints', ipKeyPoints);
AddOutput('hresult',hresult);
END_METHOD

METHOD PROTECTED OnExecute
hresult.Value := F_VN_KeyPointsFASTExp(
	ipSrcImage := ipSrcImage.Value,
    ipKeyPoints := ipKeyPoints.Value,
    ipMask := ipMask.Value,
    stParams := stParams.Value,
	hrPrev:= hrPrev.Value);
END_METHOD

METHOD PUBLIC PreExecutionCheck
VAR_INPUT
	Check : I_PreExecutionChecks;
END_VAR
Check.IsTrue(ipSrcImage.IsValid, 'ipSrcImage must contain an image');
Check.IsTrue(ipSrcImage.HasChannelCount(1), 'ipSrcImage must have 1 channel');
END_METHOD

END_FUNCTION_BLOCK

// ---- Nodes/Keypoint Features/Node_F_VN_KeyPointsGFTTExp.TcPOU
{attribute 'linkalways'} 
{attribute 'no_explicit_call' := 'This FB is a CLASS and must be accessed using methods or properties'}
{attribute 'enable_dynamic_creation'}
FUNCTION_BLOCK Node_F_VN_KeyPointsGFTTExp EXTENDS VisionNode
VAR
    ipSrcImage : _ITcVnImage;
    ipKeyPoints : _ITcVnContainer;
    ipMask : _ITcVnImage;
    stParams : _TcVnParamsGFTT;
    hrPrev : _HRESULT(S_OK);
	hresult : _HRESULT(S_OK);
END_VAR

METHOD PUBLIC  Clone : I_Node
VAR
	pNode : POINTER TO Node_F_VN_KeyPointsGFTTExp;
END_VAR
pNode := __NEW(Node_F_VN_KeyPointsGFTTExp);
Clone := pNode^;
END_METHOD

METHOD FB_init : BOOL
VAR_INPUT
	bInitRetains : BOOL; // if TRUE, the retain variables are initialized (warm start / cold start)
	bInCopyCode : BOOL;  // if TRUE, the instance afterwards gets moved into the copy code (online change)
END_VAR
AddInput('ipSrcImage', ipSrcImage);
AddInput('ipMask', ipMask);
AddInput('stParams', stParams);
AddInput('hrPrev', hrPrev);
AddOutput('ipKeyPoints', ipKeyPoints);
AddOutput('hresult',hresult);
END_METHOD

METHOD PROTECTED OnExecute
hresult.Value := F_VN_KeyPointsGFTTExp(
	ipSrcImage := ipSrcImage.Value,
    ipKeyPoints := ipKeyPoints.Value,
    ipMask := ipMask.Value,
    stParams := stParams.Value,
	hrPrev:= hrPrev.Value);
END_METHOD

METHOD PUBLIC PreExecutionCheck
VAR_INPUT
	Check : I_PreExecutionChecks;
END_VAR
Check.IsTrue(ipSrcImage.IsValid, 'ipSrcImage must contain an image');
Check.IsTrue(ipSrcImage.HasChannelCount(1), 'ipSrcImage must have 1 channel');
END_METHOD

END_FUNCTION_BLOCK

// ---- Nodes/Keypoint Features/Node_F_VN_KeyPointsGFTT.TcPOU
{attribute 'linkalways'} 
{attribute 'no_explicit_call' := 'This FB is a CLASS and must be accessed using methods or properties'}
{attribute 'enable_dynamic_creation'}
FUNCTION_BLOCK Node_F_VN_KeyPointsGFTT EXTENDS VisionNode
VAR
    ipSrcImage : _ITcVnImage;
    ipKeyPoints : _ITcVnContainer;
    hrPrev : _HRESULT(S_OK);
	hresult : _HRESULT(S_OK);
END_VAR

METHOD PUBLIC  Clone : I_Node
VAR
	pNode : POINTER TO Node_F_VN_KeyPointsGFTT;
END_VAR
pNode := __NEW(Node_F_VN_KeyPointsGFTT);
Clone := pNode^;
END_METHOD

METHOD FB_init : BOOL
VAR_INPUT
	bInitRetains : BOOL; // if TRUE, the retain variables are initialized (warm start / cold start)
	bInCopyCode : BOOL;  // if TRUE, the instance afterwards gets moved into the copy code (online change)
END_VAR
AddInput('ipSrcImage', ipSrcImage);
AddInput('hrPrev', hrPrev);
AddOutput('ipKeyPoints', ipKeyPoints);
AddOutput('hresult',hresult);
END_METHOD

METHOD PROTECTED OnExecute
hresult.Value := F_VN_KeyPointsGFTT(
	ipSrcImage := ipSrcImage.Value,
    ipKeyPoints := ipKeyPoints.Value,
	hrPrev:= hrPrev.Value);
END_METHOD

METHOD PUBLIC PreExecutionCheck
VAR_INPUT
	Check : I_PreExecutionChecks;
END_VAR
Check.IsTrue(ipSrcImage.IsValid, 'ipSrcImage must contain an image');
Check.IsTrue(ipSrcImage.HasChannelCount(1), 'ipSrcImage must have 1 channel');
END_METHOD

END_FUNCTION_BLOCK

// ---- Nodes/Keypoint Features/Node_F_VN_KeyPointsFAST.TcPOU
{attribute 'linkalways'} 
{attribute 'no_explicit_call' := 'This FB is a CLASS and must be accessed using methods or properties'}
{attribute 'enable_dynamic_creation'}
FUNCTION_BLOCK Node_F_VN_KeyPointsFAST EXTENDS VisionNode
VAR
    ipSrcImage : _ITcVnImage;
    ipKeyPoints : _ITcVnContainer;
    hrPrev : _HRESULT(S_OK);
	hresult : _HRESULT(S_OK);
END_VAR

METHOD PUBLIC  Clone : I_Node
VAR
	pNode : POINTER TO Node_F_VN_KeyPointsFAST;
END_VAR
pNode := __NEW(Node_F_VN_KeyPointsFAST);
Clone := pNode^;
END_METHOD

METHOD FB_init : BOOL
VAR_INPUT
	bInitRetains : BOOL; // if TRUE, the retain variables are initialized (warm start / cold start)
	bInCopyCode : BOOL;  // if TRUE, the instance afterwards gets moved into the copy code (online change)
END_VAR
AddInput('ipSrcImage', ipSrcImage);
AddInput('hrPrev', hrPrev);
AddOutput('ipKeyPoints', ipKeyPoints);
AddOutput('hresult',hresult);
END_METHOD

METHOD PROTECTED OnExecute
hresult.Value := F_VN_KeyPointsFAST(
	ipSrcImage := ipSrcImage.Value,
    ipKeyPoints := ipKeyPoints.Value,
	hrPrev:= hrPrev.Value);
END_METHOD

METHOD PUBLIC PreExecutionCheck
VAR_INPUT
	Check : I_PreExecutionChecks;
END_VAR
Check.IsTrue(ipSrcImage.IsValid, 'ipSrcImage must contain an image');
Check.IsTrue(ipSrcImage.HasChannelCount(1), 'ipSrcImage must have 1 channel');
END_METHOD

END_FUNCTION_BLOCK

// ---- Nodes/Keypoint Features/Node_F_VN_KeyPointsMSERExp.TcPOU
{attribute 'linkalways'} 
{attribute 'no_explicit_call' := 'This FB is a CLASS and must be accessed using methods or properties'}
{attribute 'enable_dynamic_creation'}
FUNCTION_BLOCK Node_F_VN_KeyPointsMSERExp EXTENDS VisionNode
VAR
    ipSrcImage : _ITcVnImage;
    ipKeyPoints : _ITcVnContainer;
    ipMask : _ITcVnImage;
    stParams : _TcVnParamsMSER;
    hrPrev : _HRESULT(S_OK);
	hresult : _HRESULT(S_OK);
END_VAR

METHOD PUBLIC  Clone : I_Node
VAR
	pNode : POINTER TO Node_F_VN_KeyPointsMSERExp;
END_VAR
pNode := __NEW(Node_F_VN_KeyPointsMSERExp);
Clone := pNode^;
END_METHOD

METHOD FB_init : BOOL
VAR_INPUT
	bInitRetains : BOOL; // if TRUE, the retain variables are initialized (warm start / cold start)
	bInCopyCode : BOOL;  // if TRUE, the instance afterwards gets moved into the copy code (online change)
END_VAR
AddInput('ipSrcImage', ipSrcImage);
AddInput('ipMask', ipMask);
AddInput('stParams', stParams);
AddInput('hrPrev', hrPrev);
AddOutput('ipKeyPoints', ipKeyPoints);
AddOutput('hresult',hresult);
END_METHOD

METHOD PROTECTED OnExecute
hresult.Value := F_VN_KeyPointsMSERExp(
	ipSrcImage := ipSrcImage.Value,
    ipKeyPoints := ipKeyPoints.Value,
    ipMask := ipMask.Value,
    stParams := stParams.Value,
	hrPrev:= hrPrev.Value);
END_METHOD

METHOD PUBLIC PreExecutionCheck
VAR_INPUT
	Check : I_PreExecutionChecks;
END_VAR
Check.IsTrue(ipSrcImage.IsValid, 'ipSrcImage must contain an image');
Check.IsTrue(ipSrcImage.HasChannelCount(1), 'ipSrcImage must have 1 channel');
END_METHOD

END_FUNCTION_BLOCK

// ---- Nodes/Keypoint Features/Node_F_VN_KeyPointsMSER.TcPOU
{attribute 'linkalways'} 
{attribute 'no_explicit_call' := 'This FB is a CLASS and must be accessed using methods or properties'}
{attribute 'enable_dynamic_creation'}
FUNCTION_BLOCK Node_F_VN_KeyPointsMSER EXTENDS VisionNode
VAR
    ipSrcImage : _ITcVnImage;
    ipKeyPoints : _ITcVnContainer;
    hrPrev : _HRESULT(S_OK);
	hresult : _HRESULT(S_OK);
END_VAR

METHOD PUBLIC  Clone : I_Node
VAR
	pNode : POINTER TO Node_F_VN_KeyPointsMSER;
END_VAR
pNode := __NEW(Node_F_VN_KeyPointsMSER);
Clone := pNode^;
END_METHOD

METHOD FB_init : BOOL
VAR_INPUT
	bInitRetains : BOOL; // if TRUE, the retain variables are initialized (warm start / cold start)
	bInCopyCode : BOOL;  // if TRUE, the instance afterwards gets moved into the copy code (online change)
END_VAR
AddInput('ipSrcImage', ipSrcImage);
AddInput('hrPrev', hrPrev);
AddOutput('ipKeyPoints', ipKeyPoints);
AddOutput('hresult',hresult);
END_METHOD

METHOD PROTECTED OnExecute
hresult.Value := F_VN_KeyPointsMSER(
	ipSrcImage := ipSrcImage.Value,
    ipKeyPoints := ipKeyPoints.Value,
	hrPrev:= hrPrev.Value);
END_METHOD

METHOD PUBLIC PreExecutionCheck
VAR_INPUT
	Check : I_PreExecutionChecks;
END_VAR
Check.IsTrue(ipSrcImage.IsValid, 'ipSrcImage must contain an image');
Check.IsTrue(ipSrcImage.HasChannelCount(1), 'ipSrcImage must have 1 channel');
END_METHOD

END_FUNCTION_BLOCK

// ---- Nodes/Keypoint Features/Node_F_VN_KeyPointsSBExp.TcPOU
{attribute 'linkalways'} 
{attribute 'no_explicit_call' := 'This FB is a CLASS and must be accessed using methods or properties'}
{attribute 'enable_dynamic_creation'}
FUNCTION_BLOCK Node_F_VN_KeyPointsSBExp EXTENDS VisionNode
VAR
    ipSrcImage : _ITcVnImage;
    ipKeyPoints : _ITcVnContainer;
    ipMask : _ITcVnImage;
    stParams : _TcVnParamsSB;
    hrPrev : _HRESULT(S_OK);
	hresult : _HRESULT(S_OK);
END_VAR

METHOD PUBLIC  Clone : I_Node
VAR
	pNode : POINTER TO Node_F_VN_KeyPointsSBExp;
END_VAR
pNode := __NEW(Node_F_VN_KeyPointsSBExp);
Clone := pNode^;
END_METHOD

METHOD FB_init : BOOL
VAR_INPUT
	bInitRetains : BOOL; // if TRUE, the retain variables are initialized (warm start / cold start)
	bInCopyCode : BOOL;  // if TRUE, the instance afterwards gets moved into the copy code (online change)
END_VAR
AddInput('ipSrcImage', ipSrcImage);
AddInput('ipMask', ipMask);
AddInput('stParams', stParams);
AddInput('hrPrev', hrPrev);
AddOutput('ipKeyPoints', ipKeyPoints);
AddOutput('hresult',hresult);
END_METHOD

METHOD PROTECTED OnExecute
hresult.Value := F_VN_KeyPointsSBExp(
	ipSrcImage := ipSrcImage.Value,
    ipKeyPoints := ipKeyPoints.Value,
    ipMask := ipMask.Value,
    stParams := stParams.Value,
	hrPrev:= hrPrev.Value);
END_METHOD

METHOD PUBLIC PreExecutionCheck
VAR_INPUT
	Check : I_PreExecutionChecks;
END_VAR
Check.IsTrue(ipSrcImage.IsValid, 'ipSrcImage must contain an image');
Check.IsTrue(ipSrcImage.HasChannelCount(1), 'ipSrcImage must have 1 channel');
END_METHOD

END_FUNCTION_BLOCK

// ---- Nodes/Keypoint Features/Node_F_VN_KeyPointsSB.TcPOU
{attribute 'linkalways'} 
{attribute 'no_explicit_call' := 'This FB is a CLASS and must be accessed using methods or properties'}
{attribute 'enable_dynamic_creation'}
FUNCTION_BLOCK Node_F_VN_KeyPointsSB EXTENDS VisionNode
VAR
    ipSrcImage : _ITcVnImage;
    ipKeyPoints : _ITcVnContainer;
    hrPrev : _HRESULT(S_OK);
	hresult : _HRESULT(S_OK);
END_VAR

METHOD PUBLIC  Clone : I_Node
VAR
	pNode : POINTER TO Node_F_VN_KeyPointsSB;
END_VAR
pNode := __NEW(Node_F_VN_KeyPointsSB);
Clone := pNode^;
END_METHOD

METHOD FB_init : BOOL
VAR_INPUT
	bInitRetains : BOOL; // if TRUE, the retain variables are initialized (warm start / cold start)
	bInCopyCode : BOOL;  // if TRUE, the instance afterwards gets moved into the copy code (online change)
END_VAR
AddInput('ipSrcImage', ipSrcImage);
AddInput('hrPrev', hrPrev);
AddOutput('ipKeyPoints', ipKeyPoints);
AddOutput('hresult',hresult);
END_METHOD

METHOD PROTECTED OnExecute
hresult.Value := F_VN_KeyPointsSB(
	ipSrcImage := ipSrcImage.Value,
    ipKeyPoints := ipKeyPoints.Value,
	hrPrev:= hrPrev.Value);
END_METHOD

METHOD PUBLIC PreExecutionCheck
VAR_INPUT
	Check : I_PreExecutionChecks;
END_VAR
Check.IsTrue(ipSrcImage.IsValid, 'ipSrcImage must contain an image');
Check.IsTrue(ipSrcImage.HasChannelCount(1), 'ipSrcImage must have 1 channel');
END_METHOD

END_FUNCTION_BLOCK

// ---- Nodes/VisionNodePack.TcPOU
{attribute 'linkalways'} 
{attribute 'no_explicit_call' := 'This FB is a CLASS and must be accessed using methods or properties'}
{attribute 'enable_dynamic_creation'}
FUNCTION_BLOCK VisionNodePack
VAR
    // Algebraic Container Operations
    node_F_VN_AddToContainerElements_DINT : Node_F_VN_AddToContainerElements_DINT;
    node_F_VN_AddToContainerElements_INT : Node_F_VN_AddToContainerElements_INT;
    node_F_VN_AddToContainerElements_LREAL : Node_F_VN_AddToContainerElements_LREAL;
    node_F_VN_AddToContainerElements_REAL : Node_F_VN_AddToContainerElements_REAL;
    node_F_VN_AddToContainerElements_SINT : Node_F_VN_AddToContainerElements_SINT;
    node_F_VN_AddToContainerElements_TcVnKeyPoint : Node_F_VN_AddToContainerElements_TcVnKeyPoint;
    node_F_VN_AddToContainerElements_TcVnPoint2_DINT : Node_F_VN_AddToContainerElements_TcVnPoint2_DINT;
    node_F_VN_AddToContainerElements_TcVnPoint2_LREAL : Node_F_VN_AddToContainerElements_TcVnPoint2_LREAL;
    node_F_VN_AddToContainerElements_TcVnPoint2_REAL : Node_F_VN_AddToContainerElements_TcVnPoint2_REAL;
    node_F_VN_AddToContainerElements_TcVnPoint3_LREAL : Node_F_VN_AddToContainerElements_TcVnPoint3_LREAL;
    node_F_VN_AddToContainerElements_TcVnPoint3_REAL : Node_F_VN_AddToContainerElements_TcVnPoint3_REAL;
    node_F_VN_AddToContainerElements_TcVnRectangle_DINT : Node_F_VN_AddToContainerElements_TcVnRectangle_DINT;
    node_F_VN_AddToContainerElements_TcVnRotatedRectangle : Node_F_VN_AddToContainerElements_TcVnRotatedRectangle;
    node_F_VN_AddToContainerElements_TcVnVector2_DINT : Node_F_VN_AddToContainerElements_TcVnVector2_DINT;
    node_F_VN_AddToContainerElements_TcVnVector2_INT : Node_F_VN_AddToContainerElements_TcVnVector2_INT;
    node_F_VN_AddToContainerElements_TcVnVector2_REAL : Node_F_VN_AddToContainerElements_TcVnVector2_REAL;
    node_F_VN_AddToContainerElements_TcVnVector2_SINT : Node_F_VN_AddToContainerElements_TcVnVector2_SINT;
    node_F_VN_AddToContainerElements_TcVnVector2_UINT : Node_F_VN_AddToContainerElements_TcVnVector2_UINT;
    node_F_VN_AddToContainerElements_TcVnVector2_USINT : Node_F_VN_AddToContainerElements_TcVnVector2_USINT;
    node_F_VN_AddToContainerElements_TcVnVector3_INT : Node_F_VN_AddToContainerElements_TcVnVector3_INT;
    node_F_VN_AddToContainerElements_TcVnVector3_REAL : Node_F_VN_AddToContainerElements_TcVnVector3_REAL;
    node_F_VN_AddToContainerElements_TcVnVector3_SINT : Node_F_VN_AddToContainerElements_TcVnVector3_SINT;
    node_F_VN_AddToContainerElements_TcVnVector3_UINT : Node_F_VN_AddToContainerElements_TcVnVector3_UINT;
    node_F_VN_AddToContainerElements_TcVnVector3_USINT : Node_F_VN_AddToContainerElements_TcVnVector3_USINT;
    node_F_VN_AddToContainerElements_TcVnVector4_DINT : Node_F_VN_AddToContainerElements_TcVnVector4_DINT;
    node_F_VN_AddToContainerElements_TcVnVector4_INT : Node_F_VN_AddToContainerElements_TcVnVector4_INT;
    node_F_VN_AddToContainerElements_TcVnVector4_LREAL : Node_F_VN_AddToContainerElements_TcVnVector4_LREAL;
    node_F_VN_AddToContainerElements_TcVnVector4_REAL : Node_F_VN_AddToContainerElements_TcVnVector4_REAL;
    node_F_VN_AddToContainerElements_TcVnVector4_SINT : Node_F_VN_AddToContainerElements_TcVnVector4_SINT;
    node_F_VN_AddToContainerElements_TcVnVector4_UINT : Node_F_VN_AddToContainerElements_TcVnVector4_UINT;
    node_F_VN_AddToContainerElements_TcVnVector4_USINT : Node_F_VN_AddToContainerElements_TcVnVector4_USINT;
    node_F_VN_AddToContainerElements_UDINT : Node_F_VN_AddToContainerElements_UDINT;
    node_F_VN_AddToContainerElements_UINT : node_F_VN_AddToContainerElements_UINT;
    node_F_VN_AddToContainerElements_ULINT : Node_F_VN_AddToContainerElements_ULINT;
    node_F_VN_AddToContainerElements_USINT : Node_F_VN_AddToContainerElements_USINT;
    node_F_VN_AddContainers : Node_F_VN_AddContainers;
    node_F_VN_BitwiseAndContainers : Node_F_VN_BitwiseAndContainers;
    node_F_VN_BitwiseNotContainer : Node_F_VN_BitwiseNotContainer;
    node_F_VN_BitwiseOrContainers : Node_F_VN_BitwiseOrContainers;
    node_F_VN_BitwiseXorContainers : Node_F_VN_BitwiseXorContainers;
    node_F_VN_DivideContainers : Node_F_VN_DivideContainers;
    node_F_VN_DivideContainersExp : Node_F_VN_DivideContainersExp;
    node_F_VN_MaxContainer : Node_F_VN_MaxContainer;
    node_F_VN_MinContainer : Node_F_VN_MinContainer;
    node_F_VN_MultiplyContainers : Node_F_VN_MultiplyContainers;
    //node_F_VN_MultiplyWithContainerElements1 : Node_F_VN_MultiplyWithContainerElements1;
    //node_F_VN_MultiplyWithContainerElements1 : Node_F_VN_MultiplyWithContainerElements2;
    //node_F_VN_MultiplyWithContainerElements1 : Node_F_VN_MultiplyWithContainerElements3;
    //node_F_VN_MultiplyWithContainerElements1 : Node_F_VN_MultiplyWithContainerElements4;
    node_F_VN_NegateContainer : Node_F_VN_NegateContainer;
    node_F_VN_SubtractContainers : Node_F_VN_SubtractContainers;
   
    // Algebraic Image Operations
    node_F_VN_AddImages : Node_F_VN_AddImages;
    node_F_VN_AddImagesWeighted : Node_F_VN_AddImagesWeighted;
    node_F_VN_AddImagesWeightedExp : Node_F_VN_AddImagesWeightedExp;
    node_F_VN_AddScalarToImage : Node_F_VN_AddScalarToImage;
    node_F_VN_AddVectorToImage : Node_F_VN_AddVectorToImage;
    node_F_VN_BitwiseAndImages : Node_F_VN_BitwiseAndImages;
    node_F_VN_BitwiseAndImagesExp : Node_F_VN_BitwiseAndImagesExp;
    node_F_VN_BitwiseAndScalarWithImage : Node_F_VN_BitwiseAndScalarWithImage;
    node_F_VN_BitwiseAndVectorWithImage : Node_F_VN_BitwiseAndVectorWithImage;
    node_F_VN_BitwiseNotImage : Node_F_VN_BitwiseNotImage;
    node_F_VN_BitwiseNotImageExp : Node_F_VN_BitwiseNotImageExp;
    node_F_VN_BitwiseOrImages : Node_F_VN_BitwiseOrImages;
    node_F_VN_BitwiseOrImagesExp : Node_F_VN_BitwiseOrImagesExp;
    node_F_VN_BitwiseOrScalarWithImage : Node_F_VN_BitwiseOrScalarWithImage;
    node_F_VN_BitwiseOrVectorWithImage : Node_F_VN_BitwiseOrVectorWithImage;
    node_F_VN_BitwiseXorImages : Node_F_VN_BitwiseXorImages;
    node_F_VN_BitwiseXorImagesExp : Node_F_VN_BitwiseXorImagesExp;
    node_F_VN_BitwiseXorScalarWithImage : Node_F_VN_BitwiseXorScalarWithImage;
    node_F_VN_BitwiseXorVectorWithImage : Node_F_VN_BitwiseXorVectorWithImage;
    //node_F_VN_BlendImages : Node_F_VN_BlendImages;
    node_F_VN_DivideImageByScalar : Node_F_VN_DivideImageByScalar;
    node_F_VN_DivideImageByVector : Node_F_VN_DivideImageByVector;
    node_F_VN_DivideImages : Node_F_VN_DivideImages;
    node_F_VN_DivideScalarByImage : Node_F_VN_DivideScalarByImage;
    node_F_VN_DivideVectorByImage : Node_F_VN_DivideVectorByImage;
    node_F_VN_ElementwiseExp : Node_F_VN_ElementwiseExp;
    node_F_VN_ElementwiseLog : Node_F_VN_ElementwiseLog;
    node_F_VN_MaxImage : Node_F_VN_MaxImage;
    node_F_VN_MaxImageExp : Node_F_VN_MaxImageExp;
    node_F_VN_MaxImageWithScalar : Node_F_VN_MaxImageWithScalar;
    node_F_VN_MaxImageWithScalarExp : Node_F_VN_MaxImageWithScalarExp;
    node_F_VN_MaxImageWithVector : Node_F_VN_MaxImageWithVector;
    node_F_VN_MaxImageWithVectorExp : Node_F_VN_MaxImageWithVectorExp;
    node_F_VN_MinImage : Node_F_VN_MinImage;
    node_F_VN_MinImageExp : Node_F_VN_MinImageExp;
    node_F_VN_MinImageWithScalar : Node_F_VN_MinImageWithScalar;
    node_F_VN_MinImageWithScalarExp : Node_F_VN_MinImageWithScalarExp;
    node_F_VN_MinImageWithVector : Node_F_VN_MinImageWithVector;
    node_F_VN_MinImageWithVectorExp : Node_F_VN_MinImageWithVectorExp;
    node_F_VN_MultiplyImages : Node_F_VN_MultiplyImages;
    node_F_VN_MultiplyImageWithScalar : Node_F_VN_MultiplyImageWithScalar;
    node_F_VN_MultiplyImageWithVector : Node_F_VN_MultiplyImageWithVector;
    node_F_VN_SubtractImageFromScalar : Node_F_VN_SubtractImageFromScalar;
    node_F_VN_SubtractImageFromVector : Node_F_VN_SubtractImageFromVector;
    node_F_VN_SubtractImages : Node_F_VN_SubtractImages;
    node_F_VN_SubtractScalarFromImage : Node_F_VN_SubtractScalarFromImage;
    node_F_VN_SubtractVectorFromImage : Node_F_VN_SubtractVectorFromImage;
        
    // Basic Container Operations
    node_F_VN_AppendToContainer_DINT : Node_F_VN_AppendToContainer_DINT;
    node_F_VN_AppendToContainer_INT : Node_F_VN_AppendToContainer_INT;
    node_F_VN_AppendToContainer_ITcVnContainer : Node_F_VN_AppendToContainer_ITcVnContainer;
    //node_F_VN_AppendToContainer_ITcVnForwardIterator : Node_F_VN_AppendToContainer_ITcVnForwardIterator;
    node_F_VN_AppendToContainer_ITcVnImage : Node_F_VN_AppendToContainer_ITcVnImage;
    node_F_VN_AppendToContainer_LREAL : Node_F_VN_AppendToContainer_LREAL;
    node_F_VN_AppendToContainer_REAL : Node_F_VN_AppendToContainer_REAL;
    node_F_VN_AppendToContainer_SINT : Node_F_VN_AppendToContainer_SINT;
    node_F_VN_AppendToContainer_TcVnDMatch : Node_F_VN_AppendToContainer_TcVnDMatch;
    node_F_VN_AppendToContainer_TcVnKeyPoint : Node_F_VN_AppendToContainer_TcVnKeyPoint;
    node_F_VN_AppendToContainer_TcVnPoint2_DINT : Node_F_VN_AppendToContainer_TcVnPoint2_DINT;
    node_F_VN_AppendToContainer_TcVnPoint2_LREAL : Node_F_VN_AppendToContainer_TcVnPoint2_LREAL;
    node_F_VN_AppendToContainer_TcVnPoint2_REAL : Node_F_VN_AppendToContainer_TcVnPoint2_REAL;
    node_F_VN_AppendToContainer_TcVnPoint3_LREAL : Node_F_VN_AppendToContainer_TcVnPoint3_LREAL;
    node_F_VN_AppendToContainer_TcVnPoint3_REAL : Node_F_VN_AppendToContainer_TcVnPoint3_REAL;
    node_F_VN_AppendToContainer_TcVnRectangle_DINT : Node_F_VN_AppendToContainer_TcVnRectangle_DINT;
    node_F_VN_AppendToContainer_TcVnRotatedRectangle : Node_F_VN_AppendToContainer_TcVnRotatedRectangle;
    node_F_VN_AppendToContainer_TcVnVector2_DINT : Node_F_VN_AppendToContainer_TcVnVector2_DINT;
    node_F_VN_AppendToContainer_TcVnVector2_INT : Node_F_VN_AppendToContainer_TcVnVector2_INT;
    node_F_VN_AppendToContainer_TcVnVector2_REAL : Node_F_VN_AppendToContainer_TcVnVector2_REAL;
    node_F_VN_AppendToContainer_TcVnVector2_SINT : Node_F_VN_AppendToContainer_TcVnVector2_SINT;
    node_F_VN_AppendToContainer_TcVnVector2_UINT : Node_F_VN_AppendToContainer_TcVnVector2_UINT;
    node_F_VN_AppendToContainer_TcVnVector2_USINT : Node_F_VN_AppendToContainer_TcVnVector2_USINT;
    node_F_VN_AppendToContainer_TcVnVector3_INT : Node_F_VN_AppendToContainer_TcVnVector3_INT;
    node_F_VN_AppendToContainer_TcVnVector3_REAL : Node_F_VN_AppendToContainer_TcVnVector3_REAL;
    node_F_VN_AppendToContainer_TcVnVector3_SINT : Node_F_VN_AppendToContainer_TcVnVector3_SINT;
    node_F_VN_AppendToContainer_TcVnVector3_UINT : Node_F_VN_AppendToContainer_TcVnVector3_UINT;
    node_F_VN_AppendToContainer_TcVnVector3_USINT : Node_F_VN_AppendToContainer_TcVnVector3_USINT;
    node_F_VN_AppendToContainer_TcVnVector4_DINT : Node_F_VN_AppendToContainer_TcVnVector4_DINT;
    node_F_VN_AppendToContainer_TcVnVector4_INT : Node_F_VN_AppendToContainer_TcVnVector4_INT;
    node_F_VN_AppendToContainer_TcVnVector4_LREAL : Node_F_VN_AppendToContainer_TcVnVector4_LREAL;
    node_F_VN_AppendToContainer_TcVnVector4_REAL : Node_F_VN_AppendToContainer_TcVnVector4_REAL;
    node_F_VN_AppendToContainer_TcVnVector4_SINT : Node_F_VN_AppendToContainer_TcVnVector4_SINT;
    node_F_VN_AppendToContainer_TcVnVector4_UINT : Node_F_VN_AppendToContainer_TcVnVector4_UINT;
    node_F_VN_AppendToContainer_TcVnVector4_USINT : Node_F_VN_AppendToContainer_TcVnVector4_USINT;
    node_F_VN_AppendToContainer_UDINT : Node_F_VN_AppendToContainer_UDINT;
    node_F_VN_AppendToContainer_UINT : node_F_VN_AppendToContainer_UINT;
    node_F_VN_AppendToContainer_ULINT : Node_F_VN_AppendToContainer_ULINT;
    node_F_VN_AppendToContainer_USINT : Node_F_VN_AppendToContainer_USINT;
    
